// TIA Portal V19 export
FUNCTION "MFG TRANSFER CYCLE" : Void   // FC23, LAD
{ S7_Optimized_Access := 'TRUE' }
// stored: SetENOAutomatically false
   VAR_TEMP   // added for the SCL form of the ladder/FBD networks
      _w1 : Bool;
   END_VAR
BEGIN

REGION Network 1: TRANSFER SELECT
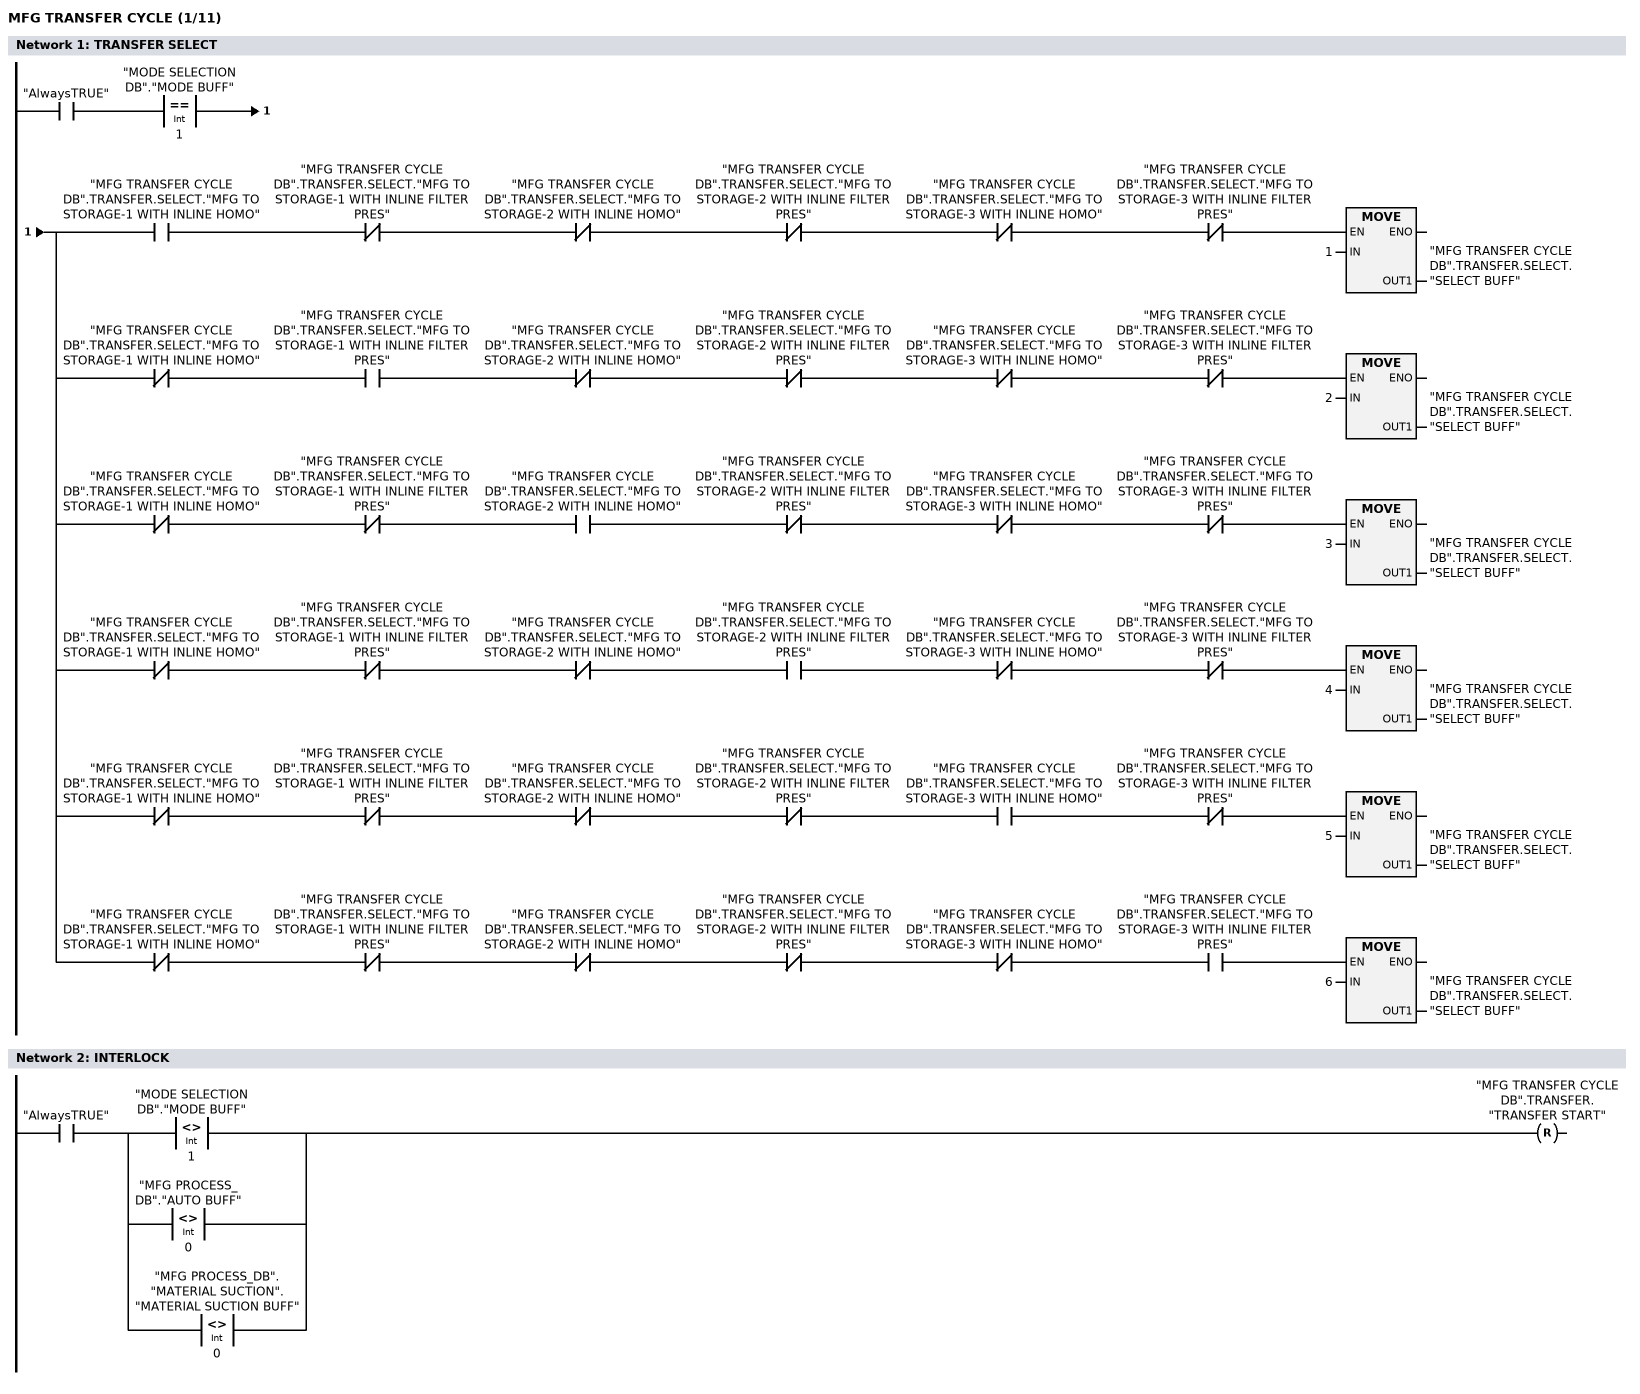
   RUNG wire#powerrail
      Contact( "AlwaysTRUE" )
      { S7_Templates := "SrcType := Int" } EQ_Contact(in1 := "MODE SELECTION DB"."MODE BUFF", in2 := 1)
      wire#w1
      Contact( "MFG TRANSFER CYCLE DB".TRANSFER.SELECT."MFG TO STORAGE-1 WITH INLINE HOMO" )
      I_Contact( "MFG TRANSFER CYCLE DB".TRANSFER.SELECT."MFG TO STORAGE-1 WITH INLINE FILTER PRES" )
      I_Contact( "MFG TRANSFER CYCLE DB".TRANSFER.SELECT."MFG TO STORAGE-2 WITH INLINE HOMO" )
      I_Contact( "MFG TRANSFER CYCLE DB".TRANSFER.SELECT."MFG TO STORAGE-2 WITH INLINE FILTER PRES" )
      I_Contact( "MFG TRANSFER CYCLE DB".TRANSFER.SELECT."MFG TO STORAGE-3 WITH INLINE HOMO" )
      I_Contact( "MFG TRANSFER CYCLE DB".TRANSFER.SELECT."MFG TO STORAGE-3 WITH INLINE FILTER PRES" )
      Move(in := 1, out1 => "MFG TRANSFER CYCLE DB".TRANSFER.SELECT."SELECT BUFF")
   END_RUNG
   RUNG wire#w1
      I_Contact( "MFG TRANSFER CYCLE DB".TRANSFER.SELECT."MFG TO STORAGE-1 WITH INLINE HOMO" )
      Contact( "MFG TRANSFER CYCLE DB".TRANSFER.SELECT."MFG TO STORAGE-1 WITH INLINE FILTER PRES" )
      I_Contact( "MFG TRANSFER CYCLE DB".TRANSFER.SELECT."MFG TO STORAGE-2 WITH INLINE HOMO" )
      I_Contact( "MFG TRANSFER CYCLE DB".TRANSFER.SELECT."MFG TO STORAGE-2 WITH INLINE FILTER PRES" )
      I_Contact( "MFG TRANSFER CYCLE DB".TRANSFER.SELECT."MFG TO STORAGE-3 WITH INLINE HOMO" )
      I_Contact( "MFG TRANSFER CYCLE DB".TRANSFER.SELECT."MFG TO STORAGE-3 WITH INLINE FILTER PRES" )
      Move(in := 2, out1 => "MFG TRANSFER CYCLE DB".TRANSFER.SELECT."SELECT BUFF")
   END_RUNG
   RUNG wire#w1
      I_Contact( "MFG TRANSFER CYCLE DB".TRANSFER.SELECT."MFG TO STORAGE-1 WITH INLINE HOMO" )
      I_Contact( "MFG TRANSFER CYCLE DB".TRANSFER.SELECT."MFG TO STORAGE-1 WITH INLINE FILTER PRES" )
      Contact( "MFG TRANSFER CYCLE DB".TRANSFER.SELECT."MFG TO STORAGE-2 WITH INLINE HOMO" )
      I_Contact( "MFG TRANSFER CYCLE DB".TRANSFER.SELECT."MFG TO STORAGE-2 WITH INLINE FILTER PRES" )
      I_Contact( "MFG TRANSFER CYCLE DB".TRANSFER.SELECT."MFG TO STORAGE-3 WITH INLINE HOMO" )
      I_Contact( "MFG TRANSFER CYCLE DB".TRANSFER.SELECT."MFG TO STORAGE-3 WITH INLINE FILTER PRES" )
      Move(in := 3, out1 => "MFG TRANSFER CYCLE DB".TRANSFER.SELECT."SELECT BUFF")
   END_RUNG
   RUNG wire#w1
      I_Contact( "MFG TRANSFER CYCLE DB".TRANSFER.SELECT."MFG TO STORAGE-1 WITH INLINE HOMO" )
      I_Contact( "MFG TRANSFER CYCLE DB".TRANSFER.SELECT."MFG TO STORAGE-1 WITH INLINE FILTER PRES" )
      I_Contact( "MFG TRANSFER CYCLE DB".TRANSFER.SELECT."MFG TO STORAGE-2 WITH INLINE HOMO" )
      Contact( "MFG TRANSFER CYCLE DB".TRANSFER.SELECT."MFG TO STORAGE-2 WITH INLINE FILTER PRES" )
      I_Contact( "MFG TRANSFER CYCLE DB".TRANSFER.SELECT."MFG TO STORAGE-3 WITH INLINE HOMO" )
      I_Contact( "MFG TRANSFER CYCLE DB".TRANSFER.SELECT."MFG TO STORAGE-3 WITH INLINE FILTER PRES" )
      Move(in := 4, out1 => "MFG TRANSFER CYCLE DB".TRANSFER.SELECT."SELECT BUFF")
   END_RUNG
   RUNG wire#w1
      I_Contact( "MFG TRANSFER CYCLE DB".TRANSFER.SELECT."MFG TO STORAGE-1 WITH INLINE HOMO" )
      I_Contact( "MFG TRANSFER CYCLE DB".TRANSFER.SELECT."MFG TO STORAGE-1 WITH INLINE FILTER PRES" )
      I_Contact( "MFG TRANSFER CYCLE DB".TRANSFER.SELECT."MFG TO STORAGE-2 WITH INLINE HOMO" )
      I_Contact( "MFG TRANSFER CYCLE DB".TRANSFER.SELECT."MFG TO STORAGE-2 WITH INLINE FILTER PRES" )
      Contact( "MFG TRANSFER CYCLE DB".TRANSFER.SELECT."MFG TO STORAGE-3 WITH INLINE HOMO" )
      I_Contact( "MFG TRANSFER CYCLE DB".TRANSFER.SELECT."MFG TO STORAGE-3 WITH INLINE FILTER PRES" )
      Move(in := 5, out1 => "MFG TRANSFER CYCLE DB".TRANSFER.SELECT."SELECT BUFF")
   END_RUNG
   RUNG wire#w1
      I_Contact( "MFG TRANSFER CYCLE DB".TRANSFER.SELECT."MFG TO STORAGE-1 WITH INLINE HOMO" )
      I_Contact( "MFG TRANSFER CYCLE DB".TRANSFER.SELECT."MFG TO STORAGE-1 WITH INLINE FILTER PRES" )
      I_Contact( "MFG TRANSFER CYCLE DB".TRANSFER.SELECT."MFG TO STORAGE-2 WITH INLINE HOMO" )
      I_Contact( "MFG TRANSFER CYCLE DB".TRANSFER.SELECT."MFG TO STORAGE-2 WITH INLINE FILTER PRES" )
      I_Contact( "MFG TRANSFER CYCLE DB".TRANSFER.SELECT."MFG TO STORAGE-3 WITH INLINE HOMO" )
      Contact( "MFG TRANSFER CYCLE DB".TRANSFER.SELECT."MFG TO STORAGE-3 WITH INLINE FILTER PRES" )
      Move(in := 6, out1 => "MFG TRANSFER CYCLE DB".TRANSFER.SELECT."SELECT BUFF")
   END_RUNG
   // the same network as SCL:
   #_w1 := "AlwaysTRUE" AND ("MODE SELECTION DB"."MODE BUFF" = 1);
   IF #_w1 AND "MFG TRANSFER CYCLE DB".TRANSFER.SELECT."MFG TO STORAGE-1 WITH INLINE HOMO" AND NOT "MFG TRANSFER CYCLE DB".TRANSFER.SELECT."MFG TO STORAGE-1 WITH INLINE FILTER PRES" AND NOT "MFG TRANSFER CYCLE DB".TRANSFER.SELECT."MFG TO STORAGE-2 WITH INLINE HOMO" AND NOT "MFG TRANSFER CYCLE DB".TRANSFER.SELECT."MFG TO STORAGE-2 WITH INLINE FILTER PRES" AND NOT "MFG TRANSFER CYCLE DB".TRANSFER.SELECT."MFG TO STORAGE-3 WITH INLINE HOMO" AND NOT "MFG TRANSFER CYCLE DB".TRANSFER.SELECT."MFG TO STORAGE-3 WITH INLINE FILTER PRES" THEN
       "MFG TRANSFER CYCLE DB".TRANSFER.SELECT."SELECT BUFF" := 1;
   END_IF;
   IF #_w1 AND NOT "MFG TRANSFER CYCLE DB".TRANSFER.SELECT."MFG TO STORAGE-1 WITH INLINE HOMO" AND "MFG TRANSFER CYCLE DB".TRANSFER.SELECT."MFG TO STORAGE-1 WITH INLINE FILTER PRES" AND NOT "MFG TRANSFER CYCLE DB".TRANSFER.SELECT."MFG TO STORAGE-2 WITH INLINE HOMO" AND NOT "MFG TRANSFER CYCLE DB".TRANSFER.SELECT."MFG TO STORAGE-2 WITH INLINE FILTER PRES" AND NOT "MFG TRANSFER CYCLE DB".TRANSFER.SELECT."MFG TO STORAGE-3 WITH INLINE HOMO" AND NOT "MFG TRANSFER CYCLE DB".TRANSFER.SELECT."MFG TO STORAGE-3 WITH INLINE FILTER PRES" THEN
       "MFG TRANSFER CYCLE DB".TRANSFER.SELECT."SELECT BUFF" := 2;
   END_IF;
   IF #_w1 AND NOT "MFG TRANSFER CYCLE DB".TRANSFER.SELECT."MFG TO STORAGE-1 WITH INLINE HOMO" AND NOT "MFG TRANSFER CYCLE DB".TRANSFER.SELECT."MFG TO STORAGE-1 WITH INLINE FILTER PRES" AND "MFG TRANSFER CYCLE DB".TRANSFER.SELECT."MFG TO STORAGE-2 WITH INLINE HOMO" AND NOT "MFG TRANSFER CYCLE DB".TRANSFER.SELECT."MFG TO STORAGE-2 WITH INLINE FILTER PRES" AND NOT "MFG TRANSFER CYCLE DB".TRANSFER.SELECT."MFG TO STORAGE-3 WITH INLINE HOMO" AND NOT "MFG TRANSFER CYCLE DB".TRANSFER.SELECT."MFG TO STORAGE-3 WITH INLINE FILTER PRES" THEN
       "MFG TRANSFER CYCLE DB".TRANSFER.SELECT."SELECT BUFF" := 3;
   END_IF;
   IF #_w1 AND NOT "MFG TRANSFER CYCLE DB".TRANSFER.SELECT."MFG TO STORAGE-1 WITH INLINE HOMO" AND NOT "MFG TRANSFER CYCLE DB".TRANSFER.SELECT."MFG TO STORAGE-1 WITH INLINE FILTER PRES" AND NOT "MFG TRANSFER CYCLE DB".TRANSFER.SELECT."MFG TO STORAGE-2 WITH INLINE HOMO" AND "MFG TRANSFER CYCLE DB".TRANSFER.SELECT."MFG TO STORAGE-2 WITH INLINE FILTER PRES" AND NOT "MFG TRANSFER CYCLE DB".TRANSFER.SELECT."MFG TO STORAGE-3 WITH INLINE HOMO" AND NOT "MFG TRANSFER CYCLE DB".TRANSFER.SELECT."MFG TO STORAGE-3 WITH INLINE FILTER PRES" THEN
       "MFG TRANSFER CYCLE DB".TRANSFER.SELECT."SELECT BUFF" := 4;
   END_IF;
   IF #_w1 AND NOT "MFG TRANSFER CYCLE DB".TRANSFER.SELECT."MFG TO STORAGE-1 WITH INLINE HOMO" AND NOT "MFG TRANSFER CYCLE DB".TRANSFER.SELECT."MFG TO STORAGE-1 WITH INLINE FILTER PRES" AND NOT "MFG TRANSFER CYCLE DB".TRANSFER.SELECT."MFG TO STORAGE-2 WITH INLINE HOMO" AND NOT "MFG TRANSFER CYCLE DB".TRANSFER.SELECT."MFG TO STORAGE-2 WITH INLINE FILTER PRES" AND "MFG TRANSFER CYCLE DB".TRANSFER.SELECT."MFG TO STORAGE-3 WITH INLINE HOMO" AND NOT "MFG TRANSFER CYCLE DB".TRANSFER.SELECT."MFG TO STORAGE-3 WITH INLINE FILTER PRES" THEN
       "MFG TRANSFER CYCLE DB".TRANSFER.SELECT."SELECT BUFF" := 5;
   END_IF;
   IF #_w1 AND NOT "MFG TRANSFER CYCLE DB".TRANSFER.SELECT."MFG TO STORAGE-1 WITH INLINE HOMO" AND NOT "MFG TRANSFER CYCLE DB".TRANSFER.SELECT."MFG TO STORAGE-1 WITH INLINE FILTER PRES" AND NOT "MFG TRANSFER CYCLE DB".TRANSFER.SELECT."MFG TO STORAGE-2 WITH INLINE HOMO" AND NOT "MFG TRANSFER CYCLE DB".TRANSFER.SELECT."MFG TO STORAGE-2 WITH INLINE FILTER PRES" AND NOT "MFG TRANSFER CYCLE DB".TRANSFER.SELECT."MFG TO STORAGE-3 WITH INLINE HOMO" AND "MFG TRANSFER CYCLE DB".TRANSFER.SELECT."MFG TO STORAGE-3 WITH INLINE FILTER PRES" THEN
       "MFG TRANSFER CYCLE DB".TRANSFER.SELECT."SELECT BUFF" := 6;
   END_IF;
END_REGION

REGION Network 2: INTERLOCK
   RUNG wire#powerrail
      Contact( "AlwaysTRUE" )
      wire#w1
      { S7_Templates := "SrcType := Int" } NE_Contact(in1 := "MODE SELECTION DB"."MODE BUFF", in2 := 1)
      wire#w2
      R_Coil( "MFG TRANSFER CYCLE DB".TRANSFER."TRANSFER START" )
   END_RUNG
   RUNG wire#w1
      { S7_Templates := "SrcType := Int" } NE_Contact(in1 := "MFG PROCESS_DB"."AUTO BUFF", in2 := 0)
   END_RUNG wire#w2
   RUNG wire#w1
      { S7_Templates := "SrcType := Int" } NE_Contact(in1 := "MFG PROCESS_DB"."MATERIAL SUCTION"."MATERIAL SUCTION BUFF", in2 := 0)
   END_RUNG wire#w2
   // the same network as SCL:
   IF "AlwaysTRUE" AND (("MODE SELECTION DB"."MODE BUFF" <> 1) OR ("MFG PROCESS_DB"."AUTO BUFF" <> 0) OR ("MFG PROCESS_DB"."MATERIAL SUCTION"."MATERIAL SUCTION BUFF" <> 0)) THEN
       "MFG TRANSFER CYCLE DB".TRANSFER."TRANSFER START" := FALSE;
   END_IF;
END_REGION

REGION Network 3: TRANSFER START ///////////////////////////// MFG TO STORAGE-1 WITH INLINE HOMO
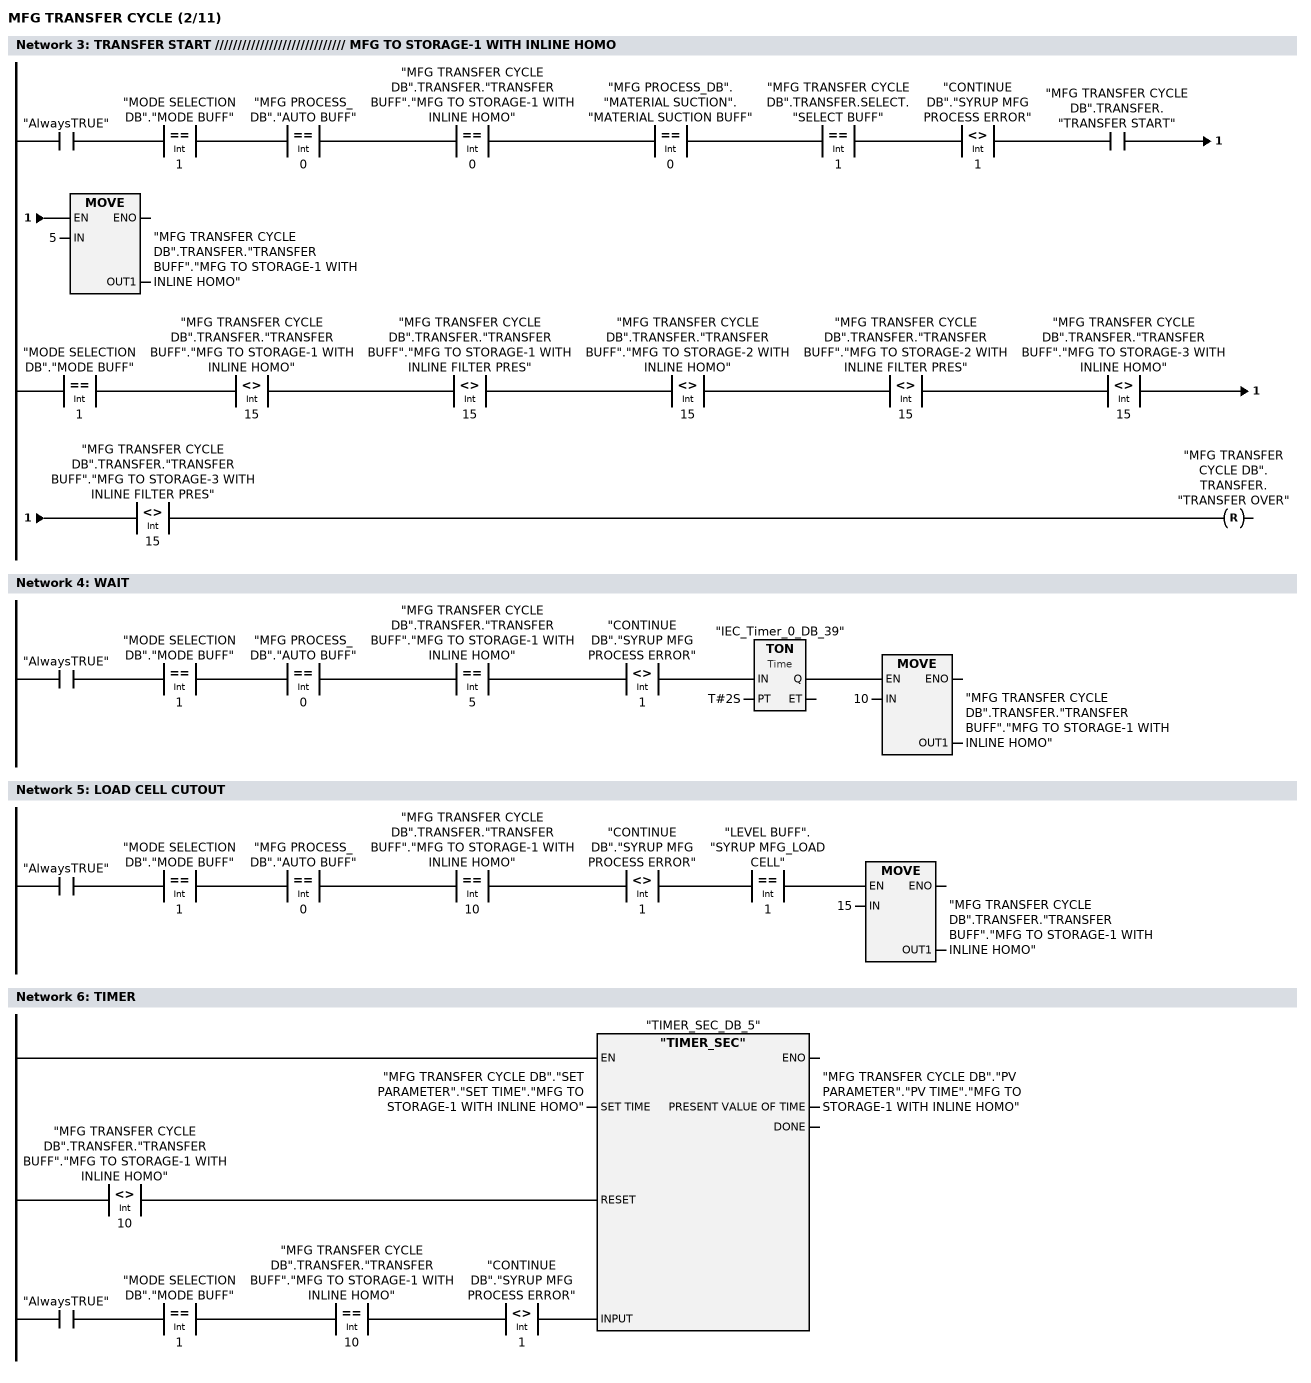
   RUNG wire#powerrail
      Contact( "AlwaysTRUE" )
      { S7_Templates := "SrcType := Int" } EQ_Contact(in1 := "MODE SELECTION DB"."MODE BUFF", in2 := 1)
      { S7_Templates := "SrcType := Int" } EQ_Contact(in1 := "MFG PROCESS_DB"."AUTO BUFF", in2 := 0)
      { S7_Templates := "SrcType := Int" } EQ_Contact(in1 := "MFG TRANSFER CYCLE DB".TRANSFER."TRANSFER BUFF"."MFG TO STORAGE-1 WITH INLINE HOMO", in2 := 0)
      { S7_Templates := "SrcType := Int" } EQ_Contact(in1 := "MFG PROCESS_DB"."MATERIAL SUCTION"."MATERIAL SUCTION BUFF", in2 := 0)
      { S7_Templates := "SrcType := Int" } EQ_Contact(in1 := "MFG TRANSFER CYCLE DB".TRANSFER.SELECT."SELECT BUFF", in2 := 1)
      { S7_Templates := "SrcType := Int" } NE_Contact(in1 := "CONTINUE DB"."SYRUP MFG PROCESS ERROR", in2 := 1)
      Contact( "MFG TRANSFER CYCLE DB".TRANSFER."TRANSFER START" )
      Move(in := 5, out1 => "MFG TRANSFER CYCLE DB".TRANSFER."TRANSFER BUFF"."MFG TO STORAGE-1 WITH INLINE HOMO")
   END_RUNG
   RUNG wire#powerrail
      { S7_Templates := "SrcType := Int" } EQ_Contact(in1 := "MODE SELECTION DB"."MODE BUFF", in2 := 1)
      { S7_Templates := "SrcType := Int" } NE_Contact(in1 := "MFG TRANSFER CYCLE DB".TRANSFER."TRANSFER BUFF"."MFG TO STORAGE-1 WITH INLINE HOMO", in2 := 15)
      { S7_Templates := "SrcType := Int" } NE_Contact(in1 := "MFG TRANSFER CYCLE DB".TRANSFER."TRANSFER BUFF"."MFG TO STORAGE-1 WITH INLINE FILTER PRES", in2 := 15)
      { S7_Templates := "SrcType := Int" } NE_Contact(in1 := "MFG TRANSFER CYCLE DB".TRANSFER."TRANSFER BUFF"."MFG TO STORAGE-2 WITH INLINE HOMO", in2 := 15)
      { S7_Templates := "SrcType := Int" } NE_Contact(in1 := "MFG TRANSFER CYCLE DB".TRANSFER."TRANSFER BUFF"."MFG TO STORAGE-2 WITH INLINE FILTER PRES", in2 := 15)
      { S7_Templates := "SrcType := Int" } NE_Contact(in1 := "MFG TRANSFER CYCLE DB".TRANSFER."TRANSFER BUFF"."MFG TO STORAGE-3 WITH INLINE HOMO", in2 := 15)
      { S7_Templates := "SrcType := Int" } NE_Contact(in1 := "MFG TRANSFER CYCLE DB".TRANSFER."TRANSFER BUFF"."MFG TO STORAGE-3 WITH INLINE FILTER PRES", in2 := 15)
      R_Coil( "MFG TRANSFER CYCLE DB".TRANSFER."TRANSFER OVER" )
   END_RUNG
   // the same network as SCL:
   IF "AlwaysTRUE" AND ("MODE SELECTION DB"."MODE BUFF" = 1) AND ("MFG PROCESS_DB"."AUTO BUFF" = 0) AND ("MFG TRANSFER CYCLE DB".TRANSFER."TRANSFER BUFF"."MFG TO STORAGE-1 WITH INLINE HOMO" = 0) AND ("MFG PROCESS_DB"."MATERIAL SUCTION"."MATERIAL SUCTION BUFF" = 0) AND ("MFG TRANSFER CYCLE DB".TRANSFER.SELECT."SELECT BUFF" = 1) AND ("CONTINUE DB"."SYRUP MFG PROCESS ERROR" <> 1) AND "MFG TRANSFER CYCLE DB".TRANSFER."TRANSFER START" THEN
       "MFG TRANSFER CYCLE DB".TRANSFER."TRANSFER BUFF"."MFG TO STORAGE-1 WITH INLINE HOMO" := 5;
   END_IF;
   IF ("MODE SELECTION DB"."MODE BUFF" = 1) AND ("MFG TRANSFER CYCLE DB".TRANSFER."TRANSFER BUFF"."MFG TO STORAGE-1 WITH INLINE HOMO" <> 15) AND ("MFG TRANSFER CYCLE DB".TRANSFER."TRANSFER BUFF"."MFG TO STORAGE-1 WITH INLINE FILTER PRES" <> 15) AND ("MFG TRANSFER CYCLE DB".TRANSFER."TRANSFER BUFF"."MFG TO STORAGE-2 WITH INLINE HOMO" <> 15) AND ("MFG TRANSFER CYCLE DB".TRANSFER."TRANSFER BUFF"."MFG TO STORAGE-2 WITH INLINE FILTER PRES" <> 15) AND ("MFG TRANSFER CYCLE DB".TRANSFER."TRANSFER BUFF"."MFG TO STORAGE-3 WITH INLINE HOMO" <> 15) AND ("MFG TRANSFER CYCLE DB".TRANSFER."TRANSFER BUFF"."MFG TO STORAGE-3 WITH INLINE FILTER PRES" <> 15) THEN
       "MFG TRANSFER CYCLE DB".TRANSFER."TRANSFER OVER" := FALSE;
   END_IF;
END_REGION

REGION Network 4: WAIT
   RUNG wire#powerrail
      Contact( "AlwaysTRUE" )
      { S7_Templates := "SrcType := Int" } EQ_Contact(in1 := "MODE SELECTION DB"."MODE BUFF", in2 := 1)
      { S7_Templates := "SrcType := Int" } EQ_Contact(in1 := "MFG PROCESS_DB"."AUTO BUFF", in2 := 0)
      { S7_Templates := "SrcType := Int" } EQ_Contact(in1 := "MFG TRANSFER CYCLE DB".TRANSFER."TRANSFER BUFF"."MFG TO STORAGE-1 WITH INLINE HOMO", in2 := 5)
      { S7_Templates := "SrcType := Int" } NE_Contact(in1 := "CONTINUE DB"."SYRUP MFG PROCESS ERROR", in2 := 1)
      { S7_Templates := "time_type := Time" } "IEC_Timer_0_DB_39".TON(pt := T#2S, et =>)
      Move(in := 10, out1 => "MFG TRANSFER CYCLE DB".TRANSFER."TRANSFER BUFF"."MFG TO STORAGE-1 WITH INLINE HOMO")
   END_RUNG
   // the same network as SCL:
   "IEC_Timer_0_DB_39".TON(IN := "AlwaysTRUE" AND ("MODE SELECTION DB"."MODE BUFF" = 1) AND ("MFG PROCESS_DB"."AUTO BUFF" = 0) AND ("MFG TRANSFER CYCLE DB".TRANSFER."TRANSFER BUFF"."MFG TO STORAGE-1 WITH INLINE HOMO" = 5) AND ("CONTINUE DB"."SYRUP MFG PROCESS ERROR" <> 1),
                           PT := T#2S);
   IF "IEC_Timer_0_DB_39".Q THEN
       "MFG TRANSFER CYCLE DB".TRANSFER."TRANSFER BUFF"."MFG TO STORAGE-1 WITH INLINE HOMO" := 10;
   END_IF;
END_REGION

REGION Network 5: LOAD CELL CUTOUT
   RUNG wire#powerrail
      Contact( "AlwaysTRUE" )
      { S7_Templates := "SrcType := Int" } EQ_Contact(in1 := "MODE SELECTION DB"."MODE BUFF", in2 := 1)
      { S7_Templates := "SrcType := Int" } EQ_Contact(in1 := "MFG PROCESS_DB"."AUTO BUFF", in2 := 0)
      { S7_Templates := "SrcType := Int" } EQ_Contact(in1 := "MFG TRANSFER CYCLE DB".TRANSFER."TRANSFER BUFF"."MFG TO STORAGE-1 WITH INLINE HOMO", in2 := 10)
      { S7_Templates := "SrcType := Int" } NE_Contact(in1 := "CONTINUE DB"."SYRUP MFG PROCESS ERROR", in2 := 1)
      { S7_Templates := "SrcType := Int" } EQ_Contact(in1 := "LEVEL BUFF"."SYRUP MFG_LOAD CELL", in2 := 1)
      Move(in := 15, out1 => "MFG TRANSFER CYCLE DB".TRANSFER."TRANSFER BUFF"."MFG TO STORAGE-1 WITH INLINE HOMO")
   END_RUNG
   // the same network as SCL:
   IF "AlwaysTRUE" AND ("MODE SELECTION DB"."MODE BUFF" = 1) AND ("MFG PROCESS_DB"."AUTO BUFF" = 0) AND ("MFG TRANSFER CYCLE DB".TRANSFER."TRANSFER BUFF"."MFG TO STORAGE-1 WITH INLINE HOMO" = 10) AND ("CONTINUE DB"."SYRUP MFG PROCESS ERROR" <> 1) AND ("LEVEL BUFF"."SYRUP MFG_LOAD CELL" = 1) THEN
       "MFG TRANSFER CYCLE DB".TRANSFER."TRANSFER BUFF"."MFG TO STORAGE-1 WITH INLINE HOMO" := 15;
   END_IF;
END_REGION

REGION Network 6: TIMER
   RUNG wire#powerrail
      "TIMER_SEC_DB_5"(RESET := wire#w1, INPUT := wire#w2, "SET TIME" := "MFG TRANSFER CYCLE DB"."SET PARAMETER"."SET TIME"."MFG TO STORAGE-1 WITH INLINE HOMO", "PRESENT VALUE OF TIME" => "MFG TRANSFER CYCLE DB"."PV PARAMETER"."PV TIME"."MFG TO STORAGE-1 WITH INLINE HOMO", DONE =>)
   END_RUNG
   RUNG wire#powerrail
      { S7_Templates := "SrcType := Int" } NE_Contact(in1 := "MFG TRANSFER CYCLE DB".TRANSFER."TRANSFER BUFF"."MFG TO STORAGE-1 WITH INLINE HOMO", in2 := 10)
   END_RUNG wire#w1
   RUNG wire#powerrail
      Contact( "AlwaysTRUE" )
      { S7_Templates := "SrcType := Int" } EQ_Contact(in1 := "MODE SELECTION DB"."MODE BUFF", in2 := 1)
      { S7_Templates := "SrcType := Int" } EQ_Contact(in1 := "MFG TRANSFER CYCLE DB".TRANSFER."TRANSFER BUFF"."MFG TO STORAGE-1 WITH INLINE HOMO", in2 := 10)
      { S7_Templates := "SrcType := Int" } NE_Contact(in1 := "CONTINUE DB"."SYRUP MFG PROCESS ERROR", in2 := 1)
   END_RUNG wire#w2
   // the same network as SCL:
   "TIMER_SEC_DB_5"("SET TIME" := "MFG TRANSFER CYCLE DB"."SET PARAMETER"."SET TIME"."MFG TO STORAGE-1 WITH INLINE HOMO",   // "TIMER_SEC"
                    RESET := "MFG TRANSFER CYCLE DB".TRANSFER."TRANSFER BUFF"."MFG TO STORAGE-1 WITH INLINE HOMO" <> 10,
                    INPUT := "AlwaysTRUE" AND ("MODE SELECTION DB"."MODE BUFF" = 1) AND ("MFG TRANSFER CYCLE DB".TRANSFER."TRANSFER BUFF"."MFG TO STORAGE-1 WITH INLINE HOMO" = 10) AND ("CONTINUE DB"."SYRUP MFG PROCESS ERROR" <> 1),
                    "PRESENT VALUE OF TIME" => "MFG TRANSFER CYCLE DB"."PV PARAMETER"."PV TIME"."MFG TO STORAGE-1 WITH INLINE HOMO");
END_REGION

REGION Network 7: TRANSFER OVER
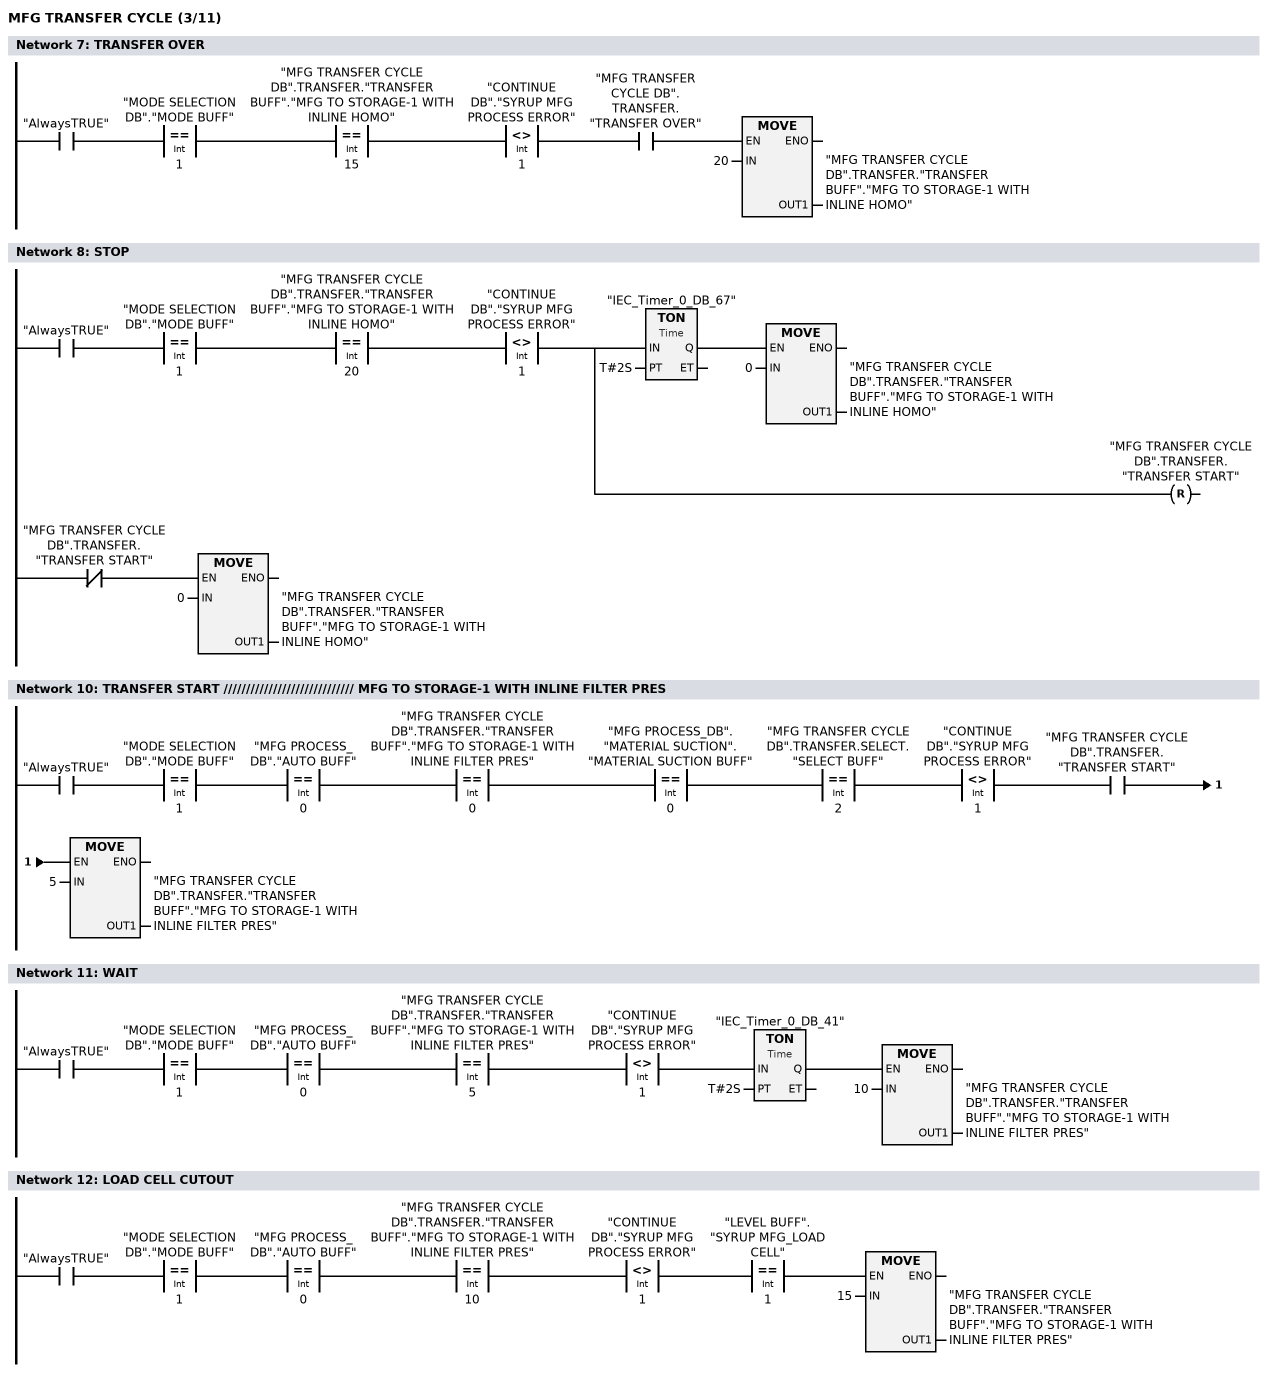
   RUNG wire#powerrail
      Contact( "AlwaysTRUE" )
      { S7_Templates := "SrcType := Int" } EQ_Contact(in1 := "MODE SELECTION DB"."MODE BUFF", in2 := 1)
      { S7_Templates := "SrcType := Int" } EQ_Contact(in1 := "MFG TRANSFER CYCLE DB".TRANSFER."TRANSFER BUFF"."MFG TO STORAGE-1 WITH INLINE HOMO", in2 := 15)
      { S7_Templates := "SrcType := Int" } NE_Contact(in1 := "CONTINUE DB"."SYRUP MFG PROCESS ERROR", in2 := 1)
      Contact( "MFG TRANSFER CYCLE DB".TRANSFER."TRANSFER OVER" )
      Move(in := 20, out1 => "MFG TRANSFER CYCLE DB".TRANSFER."TRANSFER BUFF"."MFG TO STORAGE-1 WITH INLINE HOMO")
   END_RUNG
   // the same network as SCL:
   IF "AlwaysTRUE" AND ("MODE SELECTION DB"."MODE BUFF" = 1) AND ("MFG TRANSFER CYCLE DB".TRANSFER."TRANSFER BUFF"."MFG TO STORAGE-1 WITH INLINE HOMO" = 15) AND ("CONTINUE DB"."SYRUP MFG PROCESS ERROR" <> 1) AND "MFG TRANSFER CYCLE DB".TRANSFER."TRANSFER OVER" THEN
       "MFG TRANSFER CYCLE DB".TRANSFER."TRANSFER BUFF"."MFG TO STORAGE-1 WITH INLINE HOMO" := 20;
   END_IF;
END_REGION

REGION Network 8: STOP
   RUNG wire#powerrail
      Contact( "AlwaysTRUE" )
      { S7_Templates := "SrcType := Int" } EQ_Contact(in1 := "MODE SELECTION DB"."MODE BUFF", in2 := 1)
      { S7_Templates := "SrcType := Int" } EQ_Contact(in1 := "MFG TRANSFER CYCLE DB".TRANSFER."TRANSFER BUFF"."MFG TO STORAGE-1 WITH INLINE HOMO", in2 := 20)
      { S7_Templates := "SrcType := Int" } NE_Contact(in1 := "CONTINUE DB"."SYRUP MFG PROCESS ERROR", in2 := 1)
      wire#w1
      { S7_Templates := "time_type := Time" } "IEC_Timer_0_DB_67".TON(pt := T#2S, et =>)
      Move(in := 0, out1 => "MFG TRANSFER CYCLE DB".TRANSFER."TRANSFER BUFF"."MFG TO STORAGE-1 WITH INLINE HOMO")
   END_RUNG
   RUNG wire#w1
      R_Coil( "MFG TRANSFER CYCLE DB".TRANSFER."TRANSFER START" )
   END_RUNG
   RUNG wire#powerrail
      I_Contact( "MFG TRANSFER CYCLE DB".TRANSFER."TRANSFER START" )
      Move(in := 0, out1 => "MFG TRANSFER CYCLE DB".TRANSFER."TRANSFER BUFF"."MFG TO STORAGE-1 WITH INLINE HOMO")
   END_RUNG
   // the same network as SCL:
   #_w1 := "AlwaysTRUE" AND ("MODE SELECTION DB"."MODE BUFF" = 1) AND ("MFG TRANSFER CYCLE DB".TRANSFER."TRANSFER BUFF"."MFG TO STORAGE-1 WITH INLINE HOMO" = 20) AND ("CONTINUE DB"."SYRUP MFG PROCESS ERROR" <> 1);
   "IEC_Timer_0_DB_67".TON(IN := #_w1, PT := T#2S);
   IF "IEC_Timer_0_DB_67".Q THEN
       "MFG TRANSFER CYCLE DB".TRANSFER."TRANSFER BUFF"."MFG TO STORAGE-1 WITH INLINE HOMO" := 0;
   END_IF;
   IF #_w1 THEN "MFG TRANSFER CYCLE DB".TRANSFER."TRANSFER START" := FALSE; END_IF;
   IF NOT "MFG TRANSFER CYCLE DB".TRANSFER."TRANSFER START" THEN
       "MFG TRANSFER CYCLE DB".TRANSFER."TRANSFER BUFF"."MFG TO STORAGE-1 WITH INLINE HOMO" := 0;
   END_IF;
END_REGION

REGION Network 10: TRANSFER START ///////////////////////////// MFG TO STORAGE-1 WITH INLINE FILTER PRES
   RUNG wire#powerrail
      Contact( "AlwaysTRUE" )
      { S7_Templates := "SrcType := Int" } EQ_Contact(in1 := "MODE SELECTION DB"."MODE BUFF", in2 := 1)
      { S7_Templates := "SrcType := Int" } EQ_Contact(in1 := "MFG PROCESS_DB"."AUTO BUFF", in2 := 0)
      { S7_Templates := "SrcType := Int" } EQ_Contact(in1 := "MFG TRANSFER CYCLE DB".TRANSFER."TRANSFER BUFF"."MFG TO STORAGE-1 WITH INLINE FILTER PRES", in2 := 0)
      { S7_Templates := "SrcType := Int" } EQ_Contact(in1 := "MFG PROCESS_DB"."MATERIAL SUCTION"."MATERIAL SUCTION BUFF", in2 := 0)
      { S7_Templates := "SrcType := Int" } EQ_Contact(in1 := "MFG TRANSFER CYCLE DB".TRANSFER.SELECT."SELECT BUFF", in2 := 2)
      { S7_Templates := "SrcType := Int" } NE_Contact(in1 := "CONTINUE DB"."SYRUP MFG PROCESS ERROR", in2 := 1)
      Contact( "MFG TRANSFER CYCLE DB".TRANSFER."TRANSFER START" )
      Move(in := 5, out1 => "MFG TRANSFER CYCLE DB".TRANSFER."TRANSFER BUFF"."MFG TO STORAGE-1 WITH INLINE FILTER PRES")
   END_RUNG
   // the same network as SCL:
   IF "AlwaysTRUE" AND ("MODE SELECTION DB"."MODE BUFF" = 1) AND ("MFG PROCESS_DB"."AUTO BUFF" = 0) AND ("MFG TRANSFER CYCLE DB".TRANSFER."TRANSFER BUFF"."MFG TO STORAGE-1 WITH INLINE FILTER PRES" = 0) AND ("MFG PROCESS_DB"."MATERIAL SUCTION"."MATERIAL SUCTION BUFF" = 0) AND ("MFG TRANSFER CYCLE DB".TRANSFER.SELECT."SELECT BUFF" = 2) AND ("CONTINUE DB"."SYRUP MFG PROCESS ERROR" <> 1) AND "MFG TRANSFER CYCLE DB".TRANSFER."TRANSFER START" THEN
       "MFG TRANSFER CYCLE DB".TRANSFER."TRANSFER BUFF"."MFG TO STORAGE-1 WITH INLINE FILTER PRES" := 5;
   END_IF;
END_REGION

REGION Network 11: WAIT
   RUNG wire#powerrail
      Contact( "AlwaysTRUE" )
      { S7_Templates := "SrcType := Int" } EQ_Contact(in1 := "MODE SELECTION DB"."MODE BUFF", in2 := 1)
      { S7_Templates := "SrcType := Int" } EQ_Contact(in1 := "MFG PROCESS_DB"."AUTO BUFF", in2 := 0)
      { S7_Templates := "SrcType := Int" } EQ_Contact(in1 := "MFG TRANSFER CYCLE DB".TRANSFER."TRANSFER BUFF"."MFG TO STORAGE-1 WITH INLINE FILTER PRES", in2 := 5)
      { S7_Templates := "SrcType := Int" } NE_Contact(in1 := "CONTINUE DB"."SYRUP MFG PROCESS ERROR", in2 := 1)
      { S7_Templates := "time_type := Time" } "IEC_Timer_0_DB_41".TON(pt := T#2S, et =>)
      Move(in := 10, out1 => "MFG TRANSFER CYCLE DB".TRANSFER."TRANSFER BUFF"."MFG TO STORAGE-1 WITH INLINE FILTER PRES")
   END_RUNG
   // the same network as SCL:
   "IEC_Timer_0_DB_41".TON(IN := "AlwaysTRUE" AND ("MODE SELECTION DB"."MODE BUFF" = 1) AND ("MFG PROCESS_DB"."AUTO BUFF" = 0) AND ("MFG TRANSFER CYCLE DB".TRANSFER."TRANSFER BUFF"."MFG TO STORAGE-1 WITH INLINE FILTER PRES" = 5) AND ("CONTINUE DB"."SYRUP MFG PROCESS ERROR" <> 1),
                           PT := T#2S);
   IF "IEC_Timer_0_DB_41".Q THEN
       "MFG TRANSFER CYCLE DB".TRANSFER."TRANSFER BUFF"."MFG TO STORAGE-1 WITH INLINE FILTER PRES" := 10;
   END_IF;
END_REGION

REGION Network 12: LOAD CELL CUTOUT
   RUNG wire#powerrail
      Contact( "AlwaysTRUE" )
      { S7_Templates := "SrcType := Int" } EQ_Contact(in1 := "MODE SELECTION DB"."MODE BUFF", in2 := 1)
      { S7_Templates := "SrcType := Int" } EQ_Contact(in1 := "MFG PROCESS_DB"."AUTO BUFF", in2 := 0)
      { S7_Templates := "SrcType := Int" } EQ_Contact(in1 := "MFG TRANSFER CYCLE DB".TRANSFER."TRANSFER BUFF"."MFG TO STORAGE-1 WITH INLINE FILTER PRES", in2 := 10)
      { S7_Templates := "SrcType := Int" } NE_Contact(in1 := "CONTINUE DB"."SYRUP MFG PROCESS ERROR", in2 := 1)
      { S7_Templates := "SrcType := Int" } EQ_Contact(in1 := "LEVEL BUFF"."SYRUP MFG_LOAD CELL", in2 := 1)
      Move(in := 15, out1 => "MFG TRANSFER CYCLE DB".TRANSFER."TRANSFER BUFF"."MFG TO STORAGE-1 WITH INLINE FILTER PRES")
   END_RUNG
   // the same network as SCL:
   IF "AlwaysTRUE" AND ("MODE SELECTION DB"."MODE BUFF" = 1) AND ("MFG PROCESS_DB"."AUTO BUFF" = 0) AND ("MFG TRANSFER CYCLE DB".TRANSFER."TRANSFER BUFF"."MFG TO STORAGE-1 WITH INLINE FILTER PRES" = 10) AND ("CONTINUE DB"."SYRUP MFG PROCESS ERROR" <> 1) AND ("LEVEL BUFF"."SYRUP MFG_LOAD CELL" = 1) THEN
       "MFG TRANSFER CYCLE DB".TRANSFER."TRANSFER BUFF"."MFG TO STORAGE-1 WITH INLINE FILTER PRES" := 15;
   END_IF;
END_REGION

REGION Network 13: TIMER
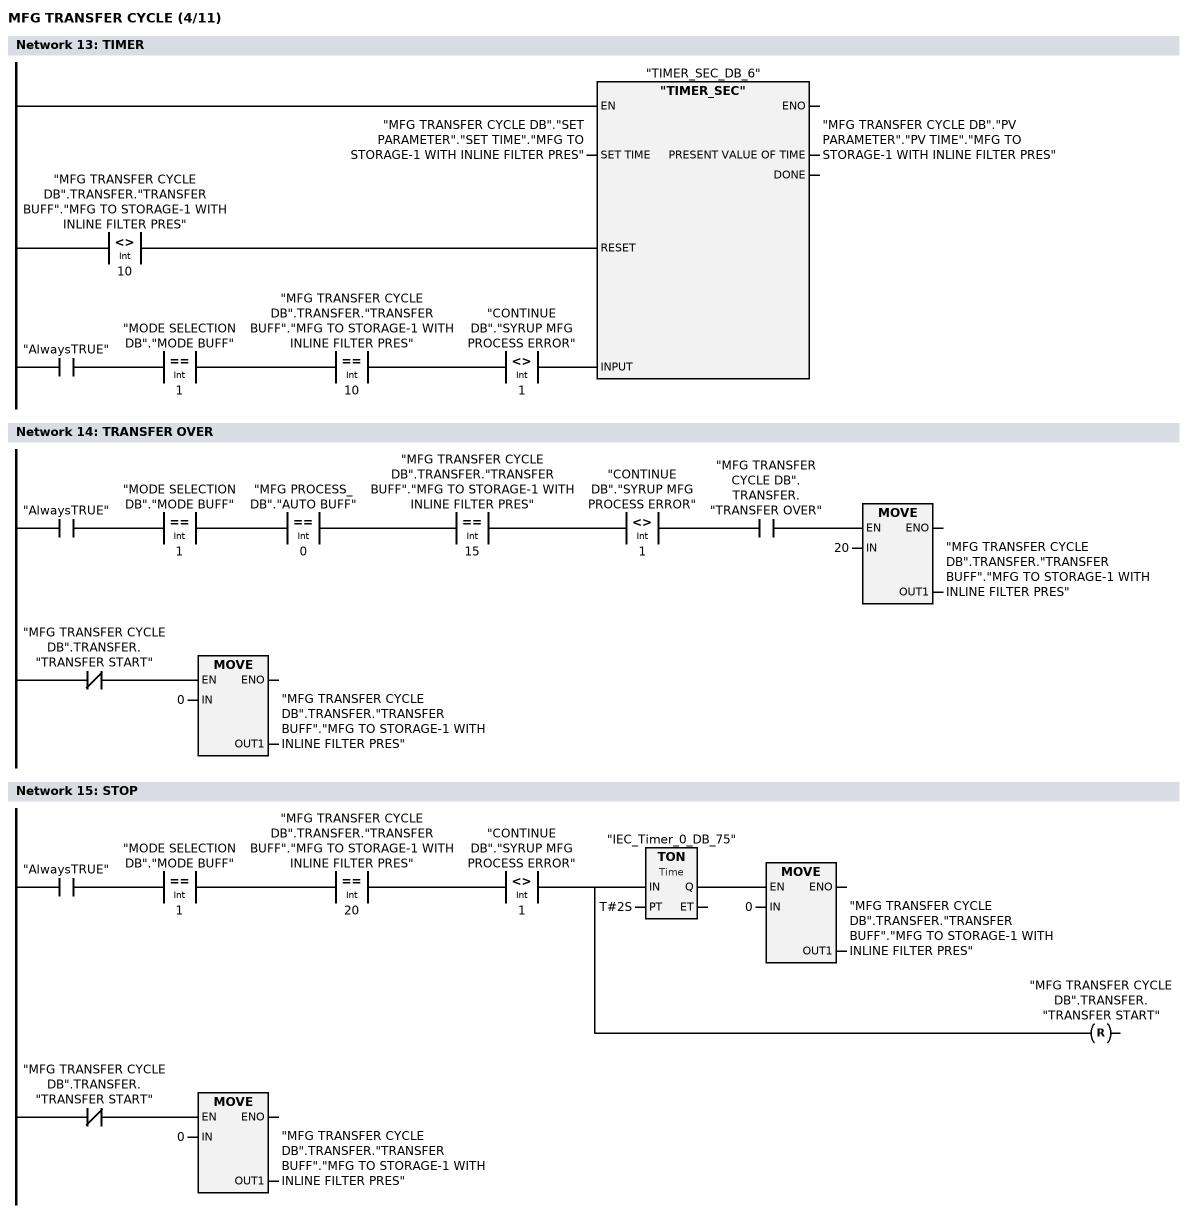
   RUNG wire#powerrail
      "TIMER_SEC_DB_6"(RESET := wire#w1, INPUT := wire#w2, "SET TIME" := "MFG TRANSFER CYCLE DB"."SET PARAMETER"."SET TIME"."MFG TO STORAGE-1 WITH INLINE FILTER PRES", "PRESENT VALUE OF TIME" => "MFG TRANSFER CYCLE DB"."PV PARAMETER"."PV TIME"."MFG TO STORAGE-1 WITH INLINE FILTER PRES", DONE =>)
   END_RUNG
   RUNG wire#powerrail
      { S7_Templates := "SrcType := Int" } NE_Contact(in1 := "MFG TRANSFER CYCLE DB".TRANSFER."TRANSFER BUFF"."MFG TO STORAGE-1 WITH INLINE FILTER PRES", in2 := 10)
   END_RUNG wire#w1
   RUNG wire#powerrail
      Contact( "AlwaysTRUE" )
      { S7_Templates := "SrcType := Int" } EQ_Contact(in1 := "MODE SELECTION DB"."MODE BUFF", in2 := 1)
      { S7_Templates := "SrcType := Int" } EQ_Contact(in1 := "MFG TRANSFER CYCLE DB".TRANSFER."TRANSFER BUFF"."MFG TO STORAGE-1 WITH INLINE FILTER PRES", in2 := 10)
      { S7_Templates := "SrcType := Int" } NE_Contact(in1 := "CONTINUE DB"."SYRUP MFG PROCESS ERROR", in2 := 1)
   END_RUNG wire#w2
   // the same network as SCL:
   "TIMER_SEC_DB_6"("SET TIME" := "MFG TRANSFER CYCLE DB"."SET PARAMETER"."SET TIME"."MFG TO STORAGE-1 WITH INLINE FILTER PRES",   // "TIMER_SEC"
                    RESET := "MFG TRANSFER CYCLE DB".TRANSFER."TRANSFER BUFF"."MFG TO STORAGE-1 WITH INLINE FILTER PRES" <> 10,
                    INPUT := "AlwaysTRUE" AND ("MODE SELECTION DB"."MODE BUFF" = 1) AND ("MFG TRANSFER CYCLE DB".TRANSFER."TRANSFER BUFF"."MFG TO STORAGE-1 WITH INLINE FILTER PRES" = 10) AND ("CONTINUE DB"."SYRUP MFG PROCESS ERROR" <> 1),
                    "PRESENT VALUE OF TIME" => "MFG TRANSFER CYCLE DB"."PV PARAMETER"."PV TIME"."MFG TO STORAGE-1 WITH INLINE FILTER PRES");
END_REGION

REGION Network 14: TRANSFER OVER
   RUNG wire#powerrail
      Contact( "AlwaysTRUE" )
      { S7_Templates := "SrcType := Int" } EQ_Contact(in1 := "MODE SELECTION DB"."MODE BUFF", in2 := 1)
      { S7_Templates := "SrcType := Int" } EQ_Contact(in1 := "MFG PROCESS_DB"."AUTO BUFF", in2 := 0)
      { S7_Templates := "SrcType := Int" } EQ_Contact(in1 := "MFG TRANSFER CYCLE DB".TRANSFER."TRANSFER BUFF"."MFG TO STORAGE-1 WITH INLINE FILTER PRES", in2 := 15)
      { S7_Templates := "SrcType := Int" } NE_Contact(in1 := "CONTINUE DB"."SYRUP MFG PROCESS ERROR", in2 := 1)
      Contact( "MFG TRANSFER CYCLE DB".TRANSFER."TRANSFER OVER" )
      Move(in := 20, out1 => "MFG TRANSFER CYCLE DB".TRANSFER."TRANSFER BUFF"."MFG TO STORAGE-1 WITH INLINE FILTER PRES")
   END_RUNG
   RUNG wire#powerrail
      I_Contact( "MFG TRANSFER CYCLE DB".TRANSFER."TRANSFER START" )
      Move(in := 0, out1 => "MFG TRANSFER CYCLE DB".TRANSFER."TRANSFER BUFF"."MFG TO STORAGE-1 WITH INLINE FILTER PRES")
   END_RUNG
   // the same network as SCL:
   IF "AlwaysTRUE" AND ("MODE SELECTION DB"."MODE BUFF" = 1) AND ("MFG PROCESS_DB"."AUTO BUFF" = 0) AND ("MFG TRANSFER CYCLE DB".TRANSFER."TRANSFER BUFF"."MFG TO STORAGE-1 WITH INLINE FILTER PRES" = 15) AND ("CONTINUE DB"."SYRUP MFG PROCESS ERROR" <> 1) AND "MFG TRANSFER CYCLE DB".TRANSFER."TRANSFER OVER" THEN
       "MFG TRANSFER CYCLE DB".TRANSFER."TRANSFER BUFF"."MFG TO STORAGE-1 WITH INLINE FILTER PRES" := 20;
   END_IF;
   IF NOT "MFG TRANSFER CYCLE DB".TRANSFER."TRANSFER START" THEN
       "MFG TRANSFER CYCLE DB".TRANSFER."TRANSFER BUFF"."MFG TO STORAGE-1 WITH INLINE FILTER PRES" := 0;
   END_IF;
END_REGION

REGION Network 15: STOP
   RUNG wire#powerrail
      Contact( "AlwaysTRUE" )
      { S7_Templates := "SrcType := Int" } EQ_Contact(in1 := "MODE SELECTION DB"."MODE BUFF", in2 := 1)
      { S7_Templates := "SrcType := Int" } EQ_Contact(in1 := "MFG TRANSFER CYCLE DB".TRANSFER."TRANSFER BUFF"."MFG TO STORAGE-1 WITH INLINE FILTER PRES", in2 := 20)
      { S7_Templates := "SrcType := Int" } NE_Contact(in1 := "CONTINUE DB"."SYRUP MFG PROCESS ERROR", in2 := 1)
      wire#w1
      { S7_Templates := "time_type := Time" } "IEC_Timer_0_DB_75".TON(pt := T#2S, et =>)
      Move(in := 0, out1 => "MFG TRANSFER CYCLE DB".TRANSFER."TRANSFER BUFF"."MFG TO STORAGE-1 WITH INLINE FILTER PRES")
   END_RUNG
   RUNG wire#w1
      R_Coil( "MFG TRANSFER CYCLE DB".TRANSFER."TRANSFER START" )
   END_RUNG
   RUNG wire#powerrail
      I_Contact( "MFG TRANSFER CYCLE DB".TRANSFER."TRANSFER START" )
      Move(in := 0, out1 => "MFG TRANSFER CYCLE DB".TRANSFER."TRANSFER BUFF"."MFG TO STORAGE-1 WITH INLINE FILTER PRES")
   END_RUNG
   // the same network as SCL:
   #_w1 := "AlwaysTRUE" AND ("MODE SELECTION DB"."MODE BUFF" = 1) AND ("MFG TRANSFER CYCLE DB".TRANSFER."TRANSFER BUFF"."MFG TO STORAGE-1 WITH INLINE FILTER PRES" = 20) AND ("CONTINUE DB"."SYRUP MFG PROCESS ERROR" <> 1);
   "IEC_Timer_0_DB_75".TON(IN := #_w1, PT := T#2S);
   IF "IEC_Timer_0_DB_75".Q THEN
       "MFG TRANSFER CYCLE DB".TRANSFER."TRANSFER BUFF"."MFG TO STORAGE-1 WITH INLINE FILTER PRES" := 0;
   END_IF;
   IF #_w1 THEN "MFG TRANSFER CYCLE DB".TRANSFER."TRANSFER START" := FALSE; END_IF;
   IF NOT "MFG TRANSFER CYCLE DB".TRANSFER."TRANSFER START" THEN
       "MFG TRANSFER CYCLE DB".TRANSFER."TRANSFER BUFF"."MFG TO STORAGE-1 WITH INLINE FILTER PRES" := 0;
   END_IF;
END_REGION

REGION Network 17: TRANSFER START ///////////////////////////// MFG TO STORAGE-2 WITH INLINE HOMO
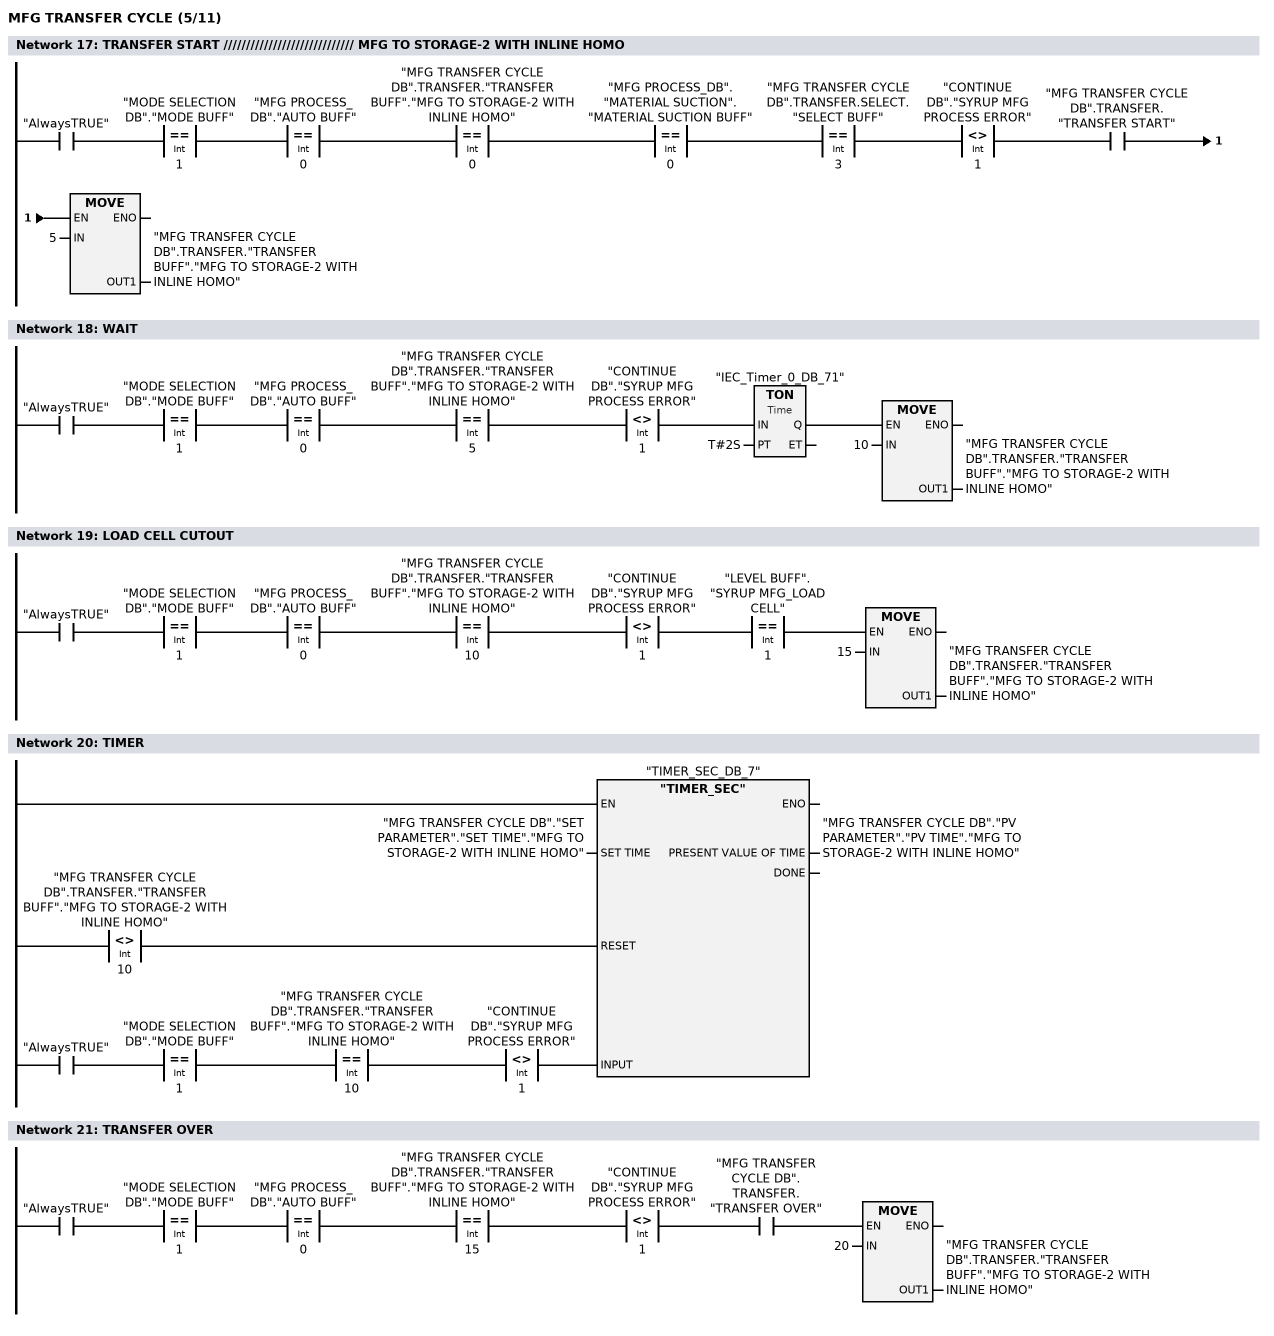
   RUNG wire#powerrail
      Contact( "AlwaysTRUE" )
      { S7_Templates := "SrcType := Int" } EQ_Contact(in1 := "MODE SELECTION DB"."MODE BUFF", in2 := 1)
      { S7_Templates := "SrcType := Int" } EQ_Contact(in1 := "MFG PROCESS_DB"."AUTO BUFF", in2 := 0)
      { S7_Templates := "SrcType := Int" } EQ_Contact(in1 := "MFG TRANSFER CYCLE DB".TRANSFER."TRANSFER BUFF"."MFG TO STORAGE-2 WITH INLINE HOMO", in2 := 0)
      { S7_Templates := "SrcType := Int" } EQ_Contact(in1 := "MFG PROCESS_DB"."MATERIAL SUCTION"."MATERIAL SUCTION BUFF", in2 := 0)
      { S7_Templates := "SrcType := Int" } EQ_Contact(in1 := "MFG TRANSFER CYCLE DB".TRANSFER.SELECT."SELECT BUFF", in2 := 3)
      { S7_Templates := "SrcType := Int" } NE_Contact(in1 := "CONTINUE DB"."SYRUP MFG PROCESS ERROR", in2 := 1)
      Contact( "MFG TRANSFER CYCLE DB".TRANSFER."TRANSFER START" )
      Move(in := 5, out1 => "MFG TRANSFER CYCLE DB".TRANSFER."TRANSFER BUFF"."MFG TO STORAGE-2 WITH INLINE HOMO")
   END_RUNG
   // the same network as SCL:
   IF "AlwaysTRUE" AND ("MODE SELECTION DB"."MODE BUFF" = 1) AND ("MFG PROCESS_DB"."AUTO BUFF" = 0) AND ("MFG TRANSFER CYCLE DB".TRANSFER."TRANSFER BUFF"."MFG TO STORAGE-2 WITH INLINE HOMO" = 0) AND ("MFG PROCESS_DB"."MATERIAL SUCTION"."MATERIAL SUCTION BUFF" = 0) AND ("MFG TRANSFER CYCLE DB".TRANSFER.SELECT."SELECT BUFF" = 3) AND ("CONTINUE DB"."SYRUP MFG PROCESS ERROR" <> 1) AND "MFG TRANSFER CYCLE DB".TRANSFER."TRANSFER START" THEN
       "MFG TRANSFER CYCLE DB".TRANSFER."TRANSFER BUFF"."MFG TO STORAGE-2 WITH INLINE HOMO" := 5;
   END_IF;
END_REGION

REGION Network 18: WAIT
   RUNG wire#powerrail
      Contact( "AlwaysTRUE" )
      { S7_Templates := "SrcType := Int" } EQ_Contact(in1 := "MODE SELECTION DB"."MODE BUFF", in2 := 1)
      { S7_Templates := "SrcType := Int" } EQ_Contact(in1 := "MFG PROCESS_DB"."AUTO BUFF", in2 := 0)
      { S7_Templates := "SrcType := Int" } EQ_Contact(in1 := "MFG TRANSFER CYCLE DB".TRANSFER."TRANSFER BUFF"."MFG TO STORAGE-2 WITH INLINE HOMO", in2 := 5)
      { S7_Templates := "SrcType := Int" } NE_Contact(in1 := "CONTINUE DB"."SYRUP MFG PROCESS ERROR", in2 := 1)
      { S7_Templates := "time_type := Time" } "IEC_Timer_0_DB_71".TON(pt := T#2S, et =>)
      Move(in := 10, out1 => "MFG TRANSFER CYCLE DB".TRANSFER."TRANSFER BUFF"."MFG TO STORAGE-2 WITH INLINE HOMO")
   END_RUNG
   // the same network as SCL:
   "IEC_Timer_0_DB_71".TON(IN := "AlwaysTRUE" AND ("MODE SELECTION DB"."MODE BUFF" = 1) AND ("MFG PROCESS_DB"."AUTO BUFF" = 0) AND ("MFG TRANSFER CYCLE DB".TRANSFER."TRANSFER BUFF"."MFG TO STORAGE-2 WITH INLINE HOMO" = 5) AND ("CONTINUE DB"."SYRUP MFG PROCESS ERROR" <> 1),
                           PT := T#2S);
   IF "IEC_Timer_0_DB_71".Q THEN
       "MFG TRANSFER CYCLE DB".TRANSFER."TRANSFER BUFF"."MFG TO STORAGE-2 WITH INLINE HOMO" := 10;
   END_IF;
END_REGION

REGION Network 19: LOAD CELL CUTOUT
   RUNG wire#powerrail
      Contact( "AlwaysTRUE" )
      { S7_Templates := "SrcType := Int" } EQ_Contact(in1 := "MODE SELECTION DB"."MODE BUFF", in2 := 1)
      { S7_Templates := "SrcType := Int" } EQ_Contact(in1 := "MFG PROCESS_DB"."AUTO BUFF", in2 := 0)
      { S7_Templates := "SrcType := Int" } EQ_Contact(in1 := "MFG TRANSFER CYCLE DB".TRANSFER."TRANSFER BUFF"."MFG TO STORAGE-2 WITH INLINE HOMO", in2 := 10)
      { S7_Templates := "SrcType := Int" } NE_Contact(in1 := "CONTINUE DB"."SYRUP MFG PROCESS ERROR", in2 := 1)
      { S7_Templates := "SrcType := Int" } EQ_Contact(in1 := "LEVEL BUFF"."SYRUP MFG_LOAD CELL", in2 := 1)
      Move(in := 15, out1 => "MFG TRANSFER CYCLE DB".TRANSFER."TRANSFER BUFF"."MFG TO STORAGE-2 WITH INLINE HOMO")
   END_RUNG
   // the same network as SCL:
   IF "AlwaysTRUE" AND ("MODE SELECTION DB"."MODE BUFF" = 1) AND ("MFG PROCESS_DB"."AUTO BUFF" = 0) AND ("MFG TRANSFER CYCLE DB".TRANSFER."TRANSFER BUFF"."MFG TO STORAGE-2 WITH INLINE HOMO" = 10) AND ("CONTINUE DB"."SYRUP MFG PROCESS ERROR" <> 1) AND ("LEVEL BUFF"."SYRUP MFG_LOAD CELL" = 1) THEN
       "MFG TRANSFER CYCLE DB".TRANSFER."TRANSFER BUFF"."MFG TO STORAGE-2 WITH INLINE HOMO" := 15;
   END_IF;
END_REGION

REGION Network 20: TIMER
   RUNG wire#powerrail
      "TIMER_SEC_DB_7"(RESET := wire#w1, INPUT := wire#w2, "SET TIME" := "MFG TRANSFER CYCLE DB"."SET PARAMETER"."SET TIME"."MFG TO STORAGE-2 WITH INLINE HOMO", "PRESENT VALUE OF TIME" => "MFG TRANSFER CYCLE DB"."PV PARAMETER"."PV TIME"."MFG TO STORAGE-2 WITH INLINE HOMO", DONE =>)
   END_RUNG
   RUNG wire#powerrail
      { S7_Templates := "SrcType := Int" } NE_Contact(in1 := "MFG TRANSFER CYCLE DB".TRANSFER."TRANSFER BUFF"."MFG TO STORAGE-2 WITH INLINE HOMO", in2 := 10)
   END_RUNG wire#w1
   RUNG wire#powerrail
      Contact( "AlwaysTRUE" )
      { S7_Templates := "SrcType := Int" } EQ_Contact(in1 := "MODE SELECTION DB"."MODE BUFF", in2 := 1)
      { S7_Templates := "SrcType := Int" } EQ_Contact(in1 := "MFG TRANSFER CYCLE DB".TRANSFER."TRANSFER BUFF"."MFG TO STORAGE-2 WITH INLINE HOMO", in2 := 10)
      { S7_Templates := "SrcType := Int" } NE_Contact(in1 := "CONTINUE DB"."SYRUP MFG PROCESS ERROR", in2 := 1)
   END_RUNG wire#w2
   // the same network as SCL:
   "TIMER_SEC_DB_7"("SET TIME" := "MFG TRANSFER CYCLE DB"."SET PARAMETER"."SET TIME"."MFG TO STORAGE-2 WITH INLINE HOMO",   // "TIMER_SEC"
                    RESET := "MFG TRANSFER CYCLE DB".TRANSFER."TRANSFER BUFF"."MFG TO STORAGE-2 WITH INLINE HOMO" <> 10,
                    INPUT := "AlwaysTRUE" AND ("MODE SELECTION DB"."MODE BUFF" = 1) AND ("MFG TRANSFER CYCLE DB".TRANSFER."TRANSFER BUFF"."MFG TO STORAGE-2 WITH INLINE HOMO" = 10) AND ("CONTINUE DB"."SYRUP MFG PROCESS ERROR" <> 1),
                    "PRESENT VALUE OF TIME" => "MFG TRANSFER CYCLE DB"."PV PARAMETER"."PV TIME"."MFG TO STORAGE-2 WITH INLINE HOMO");
END_REGION

REGION Network 21: TRANSFER OVER
   RUNG wire#powerrail
      Contact( "AlwaysTRUE" )
      { S7_Templates := "SrcType := Int" } EQ_Contact(in1 := "MODE SELECTION DB"."MODE BUFF", in2 := 1)
      { S7_Templates := "SrcType := Int" } EQ_Contact(in1 := "MFG PROCESS_DB"."AUTO BUFF", in2 := 0)
      { S7_Templates := "SrcType := Int" } EQ_Contact(in1 := "MFG TRANSFER CYCLE DB".TRANSFER."TRANSFER BUFF"."MFG TO STORAGE-2 WITH INLINE HOMO", in2 := 15)
      { S7_Templates := "SrcType := Int" } NE_Contact(in1 := "CONTINUE DB"."SYRUP MFG PROCESS ERROR", in2 := 1)
      Contact( "MFG TRANSFER CYCLE DB".TRANSFER."TRANSFER OVER" )
      Move(in := 20, out1 => "MFG TRANSFER CYCLE DB".TRANSFER."TRANSFER BUFF"."MFG TO STORAGE-2 WITH INLINE HOMO")
   END_RUNG
   // the same network as SCL:
   IF "AlwaysTRUE" AND ("MODE SELECTION DB"."MODE BUFF" = 1) AND ("MFG PROCESS_DB"."AUTO BUFF" = 0) AND ("MFG TRANSFER CYCLE DB".TRANSFER."TRANSFER BUFF"."MFG TO STORAGE-2 WITH INLINE HOMO" = 15) AND ("CONTINUE DB"."SYRUP MFG PROCESS ERROR" <> 1) AND "MFG TRANSFER CYCLE DB".TRANSFER."TRANSFER OVER" THEN
       "MFG TRANSFER CYCLE DB".TRANSFER."TRANSFER BUFF"."MFG TO STORAGE-2 WITH INLINE HOMO" := 20;
   END_IF;
END_REGION

REGION Network 22: STOP
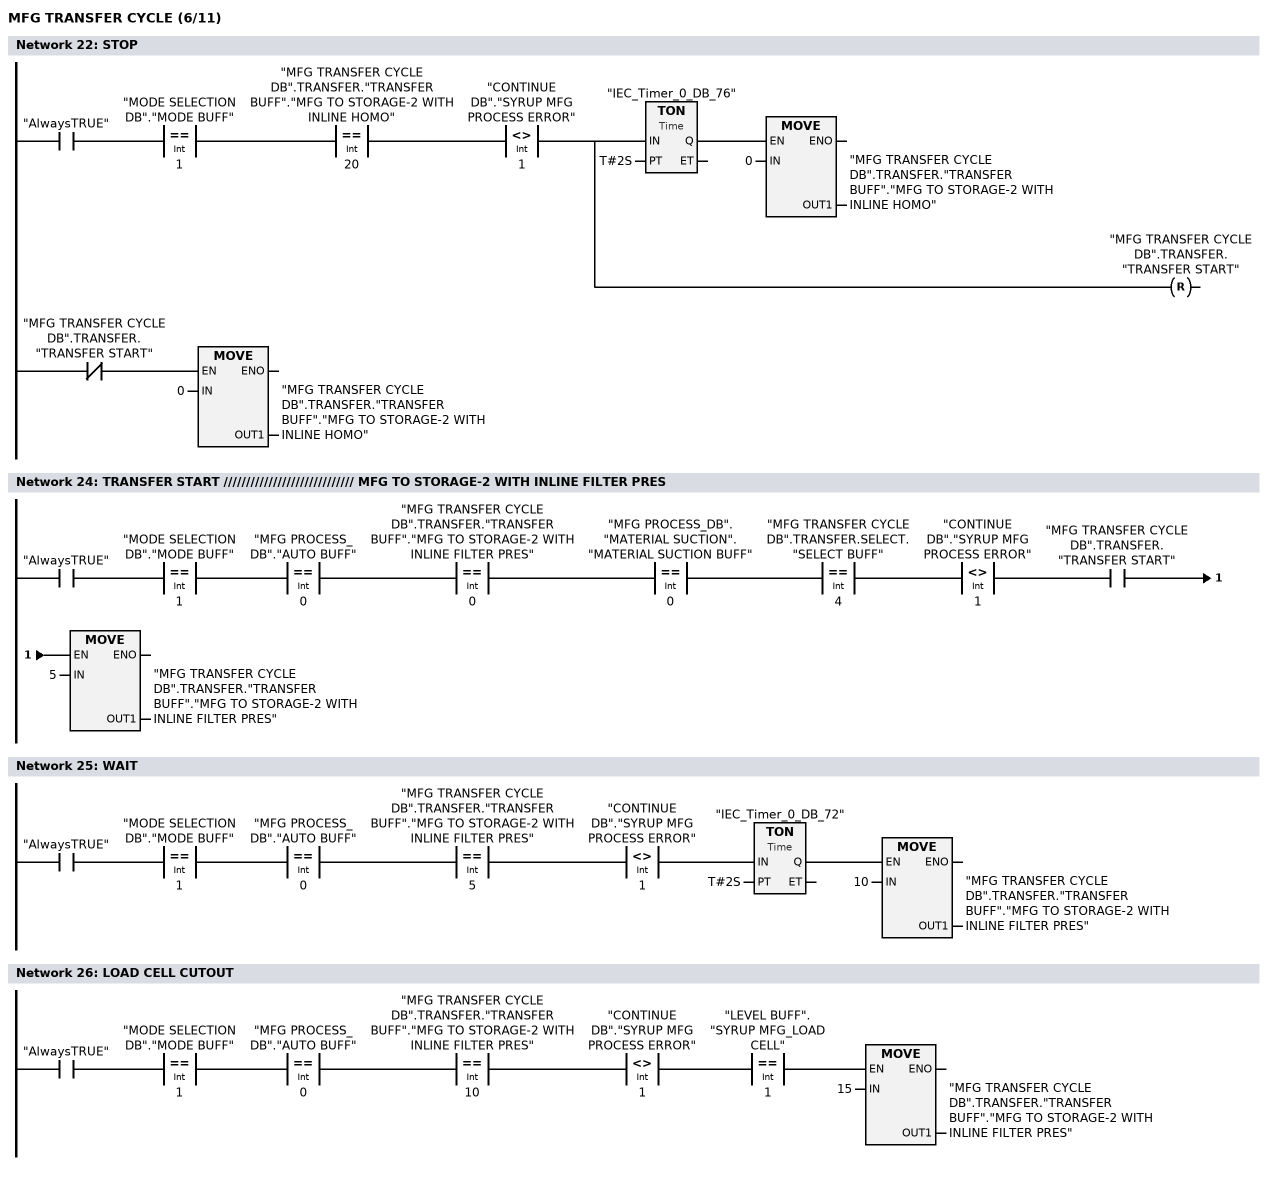
   RUNG wire#powerrail
      Contact( "AlwaysTRUE" )
      { S7_Templates := "SrcType := Int" } EQ_Contact(in1 := "MODE SELECTION DB"."MODE BUFF", in2 := 1)
      { S7_Templates := "SrcType := Int" } EQ_Contact(in1 := "MFG TRANSFER CYCLE DB".TRANSFER."TRANSFER BUFF"."MFG TO STORAGE-2 WITH INLINE HOMO", in2 := 20)
      { S7_Templates := "SrcType := Int" } NE_Contact(in1 := "CONTINUE DB"."SYRUP MFG PROCESS ERROR", in2 := 1)
      wire#w1
      { S7_Templates := "time_type := Time" } "IEC_Timer_0_DB_76".TON(pt := T#2S, et =>)
      Move(in := 0, out1 => "MFG TRANSFER CYCLE DB".TRANSFER."TRANSFER BUFF"."MFG TO STORAGE-2 WITH INLINE HOMO")
   END_RUNG
   RUNG wire#w1
      R_Coil( "MFG TRANSFER CYCLE DB".TRANSFER."TRANSFER START" )
   END_RUNG
   RUNG wire#powerrail
      I_Contact( "MFG TRANSFER CYCLE DB".TRANSFER."TRANSFER START" )
      Move(in := 0, out1 => "MFG TRANSFER CYCLE DB".TRANSFER."TRANSFER BUFF"."MFG TO STORAGE-2 WITH INLINE HOMO")
   END_RUNG
   // the same network as SCL:
   #_w1 := "AlwaysTRUE" AND ("MODE SELECTION DB"."MODE BUFF" = 1) AND ("MFG TRANSFER CYCLE DB".TRANSFER."TRANSFER BUFF"."MFG TO STORAGE-2 WITH INLINE HOMO" = 20) AND ("CONTINUE DB"."SYRUP MFG PROCESS ERROR" <> 1);
   "IEC_Timer_0_DB_76".TON(IN := #_w1, PT := T#2S);
   IF "IEC_Timer_0_DB_76".Q THEN
       "MFG TRANSFER CYCLE DB".TRANSFER."TRANSFER BUFF"."MFG TO STORAGE-2 WITH INLINE HOMO" := 0;
   END_IF;
   IF #_w1 THEN "MFG TRANSFER CYCLE DB".TRANSFER."TRANSFER START" := FALSE; END_IF;
   IF NOT "MFG TRANSFER CYCLE DB".TRANSFER."TRANSFER START" THEN
       "MFG TRANSFER CYCLE DB".TRANSFER."TRANSFER BUFF"."MFG TO STORAGE-2 WITH INLINE HOMO" := 0;
   END_IF;
END_REGION

REGION Network 24: TRANSFER START ///////////////////////////// MFG TO STORAGE-2 WITH INLINE FILTER PRES
   RUNG wire#powerrail
      Contact( "AlwaysTRUE" )
      { S7_Templates := "SrcType := Int" } EQ_Contact(in1 := "MODE SELECTION DB"."MODE BUFF", in2 := 1)
      { S7_Templates := "SrcType := Int" } EQ_Contact(in1 := "MFG PROCESS_DB"."AUTO BUFF", in2 := 0)
      { S7_Templates := "SrcType := Int" } EQ_Contact(in1 := "MFG TRANSFER CYCLE DB".TRANSFER."TRANSFER BUFF"."MFG TO STORAGE-2 WITH INLINE FILTER PRES", in2 := 0)
      { S7_Templates := "SrcType := Int" } EQ_Contact(in1 := "MFG PROCESS_DB"."MATERIAL SUCTION"."MATERIAL SUCTION BUFF", in2 := 0)
      { S7_Templates := "SrcType := Int" } EQ_Contact(in1 := "MFG TRANSFER CYCLE DB".TRANSFER.SELECT."SELECT BUFF", in2 := 4)
      { S7_Templates := "SrcType := Int" } NE_Contact(in1 := "CONTINUE DB"."SYRUP MFG PROCESS ERROR", in2 := 1)
      Contact( "MFG TRANSFER CYCLE DB".TRANSFER."TRANSFER START" )
      Move(in := 5, out1 => "MFG TRANSFER CYCLE DB".TRANSFER."TRANSFER BUFF"."MFG TO STORAGE-2 WITH INLINE FILTER PRES")
   END_RUNG
   // the same network as SCL:
   IF "AlwaysTRUE" AND ("MODE SELECTION DB"."MODE BUFF" = 1) AND ("MFG PROCESS_DB"."AUTO BUFF" = 0) AND ("MFG TRANSFER CYCLE DB".TRANSFER."TRANSFER BUFF"."MFG TO STORAGE-2 WITH INLINE FILTER PRES" = 0) AND ("MFG PROCESS_DB"."MATERIAL SUCTION"."MATERIAL SUCTION BUFF" = 0) AND ("MFG TRANSFER CYCLE DB".TRANSFER.SELECT."SELECT BUFF" = 4) AND ("CONTINUE DB"."SYRUP MFG PROCESS ERROR" <> 1) AND "MFG TRANSFER CYCLE DB".TRANSFER."TRANSFER START" THEN
       "MFG TRANSFER CYCLE DB".TRANSFER."TRANSFER BUFF"."MFG TO STORAGE-2 WITH INLINE FILTER PRES" := 5;
   END_IF;
END_REGION

REGION Network 25: WAIT
   RUNG wire#powerrail
      Contact( "AlwaysTRUE" )
      { S7_Templates := "SrcType := Int" } EQ_Contact(in1 := "MODE SELECTION DB"."MODE BUFF", in2 := 1)
      { S7_Templates := "SrcType := Int" } EQ_Contact(in1 := "MFG PROCESS_DB"."AUTO BUFF", in2 := 0)
      { S7_Templates := "SrcType := Int" } EQ_Contact(in1 := "MFG TRANSFER CYCLE DB".TRANSFER."TRANSFER BUFF"."MFG TO STORAGE-2 WITH INLINE FILTER PRES", in2 := 5)
      { S7_Templates := "SrcType := Int" } NE_Contact(in1 := "CONTINUE DB"."SYRUP MFG PROCESS ERROR", in2 := 1)
      { S7_Templates := "time_type := Time" } "IEC_Timer_0_DB_72".TON(pt := T#2S, et =>)
      Move(in := 10, out1 => "MFG TRANSFER CYCLE DB".TRANSFER."TRANSFER BUFF"."MFG TO STORAGE-2 WITH INLINE FILTER PRES")
   END_RUNG
   // the same network as SCL:
   "IEC_Timer_0_DB_72".TON(IN := "AlwaysTRUE" AND ("MODE SELECTION DB"."MODE BUFF" = 1) AND ("MFG PROCESS_DB"."AUTO BUFF" = 0) AND ("MFG TRANSFER CYCLE DB".TRANSFER."TRANSFER BUFF"."MFG TO STORAGE-2 WITH INLINE FILTER PRES" = 5) AND ("CONTINUE DB"."SYRUP MFG PROCESS ERROR" <> 1),
                           PT := T#2S);
   IF "IEC_Timer_0_DB_72".Q THEN
       "MFG TRANSFER CYCLE DB".TRANSFER."TRANSFER BUFF"."MFG TO STORAGE-2 WITH INLINE FILTER PRES" := 10;
   END_IF;
END_REGION

REGION Network 26: LOAD CELL CUTOUT
   RUNG wire#powerrail
      Contact( "AlwaysTRUE" )
      { S7_Templates := "SrcType := Int" } EQ_Contact(in1 := "MODE SELECTION DB"."MODE BUFF", in2 := 1)
      { S7_Templates := "SrcType := Int" } EQ_Contact(in1 := "MFG PROCESS_DB"."AUTO BUFF", in2 := 0)
      { S7_Templates := "SrcType := Int" } EQ_Contact(in1 := "MFG TRANSFER CYCLE DB".TRANSFER."TRANSFER BUFF"."MFG TO STORAGE-2 WITH INLINE FILTER PRES", in2 := 10)
      { S7_Templates := "SrcType := Int" } NE_Contact(in1 := "CONTINUE DB"."SYRUP MFG PROCESS ERROR", in2 := 1)
      { S7_Templates := "SrcType := Int" } EQ_Contact(in1 := "LEVEL BUFF"."SYRUP MFG_LOAD CELL", in2 := 1)
      Move(in := 15, out1 => "MFG TRANSFER CYCLE DB".TRANSFER."TRANSFER BUFF"."MFG TO STORAGE-2 WITH INLINE FILTER PRES")
   END_RUNG
   // the same network as SCL:
   IF "AlwaysTRUE" AND ("MODE SELECTION DB"."MODE BUFF" = 1) AND ("MFG PROCESS_DB"."AUTO BUFF" = 0) AND ("MFG TRANSFER CYCLE DB".TRANSFER."TRANSFER BUFF"."MFG TO STORAGE-2 WITH INLINE FILTER PRES" = 10) AND ("CONTINUE DB"."SYRUP MFG PROCESS ERROR" <> 1) AND ("LEVEL BUFF"."SYRUP MFG_LOAD CELL" = 1) THEN
       "MFG TRANSFER CYCLE DB".TRANSFER."TRANSFER BUFF"."MFG TO STORAGE-2 WITH INLINE FILTER PRES" := 15;
   END_IF;
END_REGION

REGION Network 27: TIMER
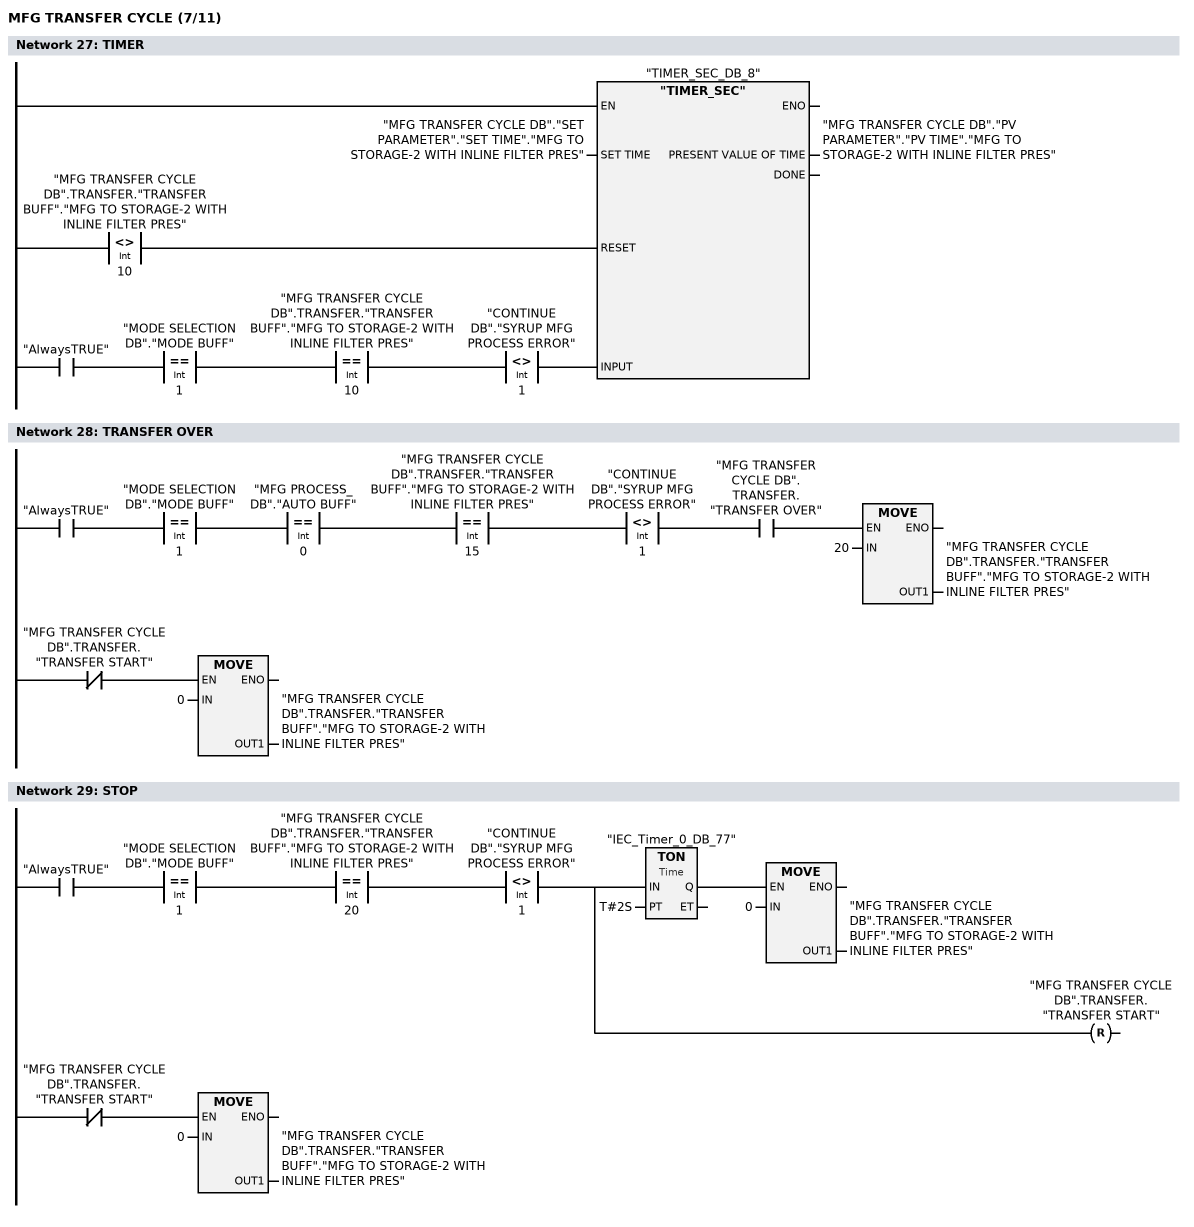
   RUNG wire#powerrail
      "TIMER_SEC_DB_8"(RESET := wire#w1, INPUT := wire#w2, "SET TIME" := "MFG TRANSFER CYCLE DB"."SET PARAMETER"."SET TIME"."MFG TO STORAGE-2 WITH INLINE FILTER PRES", "PRESENT VALUE OF TIME" => "MFG TRANSFER CYCLE DB"."PV PARAMETER"."PV TIME"."MFG TO STORAGE-2 WITH INLINE FILTER PRES", DONE =>)
   END_RUNG
   RUNG wire#powerrail
      { S7_Templates := "SrcType := Int" } NE_Contact(in1 := "MFG TRANSFER CYCLE DB".TRANSFER."TRANSFER BUFF"."MFG TO STORAGE-2 WITH INLINE FILTER PRES", in2 := 10)
   END_RUNG wire#w1
   RUNG wire#powerrail
      Contact( "AlwaysTRUE" )
      { S7_Templates := "SrcType := Int" } EQ_Contact(in1 := "MODE SELECTION DB"."MODE BUFF", in2 := 1)
      { S7_Templates := "SrcType := Int" } EQ_Contact(in1 := "MFG TRANSFER CYCLE DB".TRANSFER."TRANSFER BUFF"."MFG TO STORAGE-2 WITH INLINE FILTER PRES", in2 := 10)
      { S7_Templates := "SrcType := Int" } NE_Contact(in1 := "CONTINUE DB"."SYRUP MFG PROCESS ERROR", in2 := 1)
   END_RUNG wire#w2
   // the same network as SCL:
   "TIMER_SEC_DB_8"("SET TIME" := "MFG TRANSFER CYCLE DB"."SET PARAMETER"."SET TIME"."MFG TO STORAGE-2 WITH INLINE FILTER PRES",   // "TIMER_SEC"
                    RESET := "MFG TRANSFER CYCLE DB".TRANSFER."TRANSFER BUFF"."MFG TO STORAGE-2 WITH INLINE FILTER PRES" <> 10,
                    INPUT := "AlwaysTRUE" AND ("MODE SELECTION DB"."MODE BUFF" = 1) AND ("MFG TRANSFER CYCLE DB".TRANSFER."TRANSFER BUFF"."MFG TO STORAGE-2 WITH INLINE FILTER PRES" = 10) AND ("CONTINUE DB"."SYRUP MFG PROCESS ERROR" <> 1),
                    "PRESENT VALUE OF TIME" => "MFG TRANSFER CYCLE DB"."PV PARAMETER"."PV TIME"."MFG TO STORAGE-2 WITH INLINE FILTER PRES");
END_REGION

REGION Network 28: TRANSFER OVER
   RUNG wire#powerrail
      Contact( "AlwaysTRUE" )
      { S7_Templates := "SrcType := Int" } EQ_Contact(in1 := "MODE SELECTION DB"."MODE BUFF", in2 := 1)
      { S7_Templates := "SrcType := Int" } EQ_Contact(in1 := "MFG PROCESS_DB"."AUTO BUFF", in2 := 0)
      { S7_Templates := "SrcType := Int" } EQ_Contact(in1 := "MFG TRANSFER CYCLE DB".TRANSFER."TRANSFER BUFF"."MFG TO STORAGE-2 WITH INLINE FILTER PRES", in2 := 15)
      { S7_Templates := "SrcType := Int" } NE_Contact(in1 := "CONTINUE DB"."SYRUP MFG PROCESS ERROR", in2 := 1)
      Contact( "MFG TRANSFER CYCLE DB".TRANSFER."TRANSFER OVER" )
      Move(in := 20, out1 => "MFG TRANSFER CYCLE DB".TRANSFER."TRANSFER BUFF"."MFG TO STORAGE-2 WITH INLINE FILTER PRES")
   END_RUNG
   RUNG wire#powerrail
      I_Contact( "MFG TRANSFER CYCLE DB".TRANSFER."TRANSFER START" )
      Move(in := 0, out1 => "MFG TRANSFER CYCLE DB".TRANSFER."TRANSFER BUFF"."MFG TO STORAGE-2 WITH INLINE FILTER PRES")
   END_RUNG
   // the same network as SCL:
   IF "AlwaysTRUE" AND ("MODE SELECTION DB"."MODE BUFF" = 1) AND ("MFG PROCESS_DB"."AUTO BUFF" = 0) AND ("MFG TRANSFER CYCLE DB".TRANSFER."TRANSFER BUFF"."MFG TO STORAGE-2 WITH INLINE FILTER PRES" = 15) AND ("CONTINUE DB"."SYRUP MFG PROCESS ERROR" <> 1) AND "MFG TRANSFER CYCLE DB".TRANSFER."TRANSFER OVER" THEN
       "MFG TRANSFER CYCLE DB".TRANSFER."TRANSFER BUFF"."MFG TO STORAGE-2 WITH INLINE FILTER PRES" := 20;
   END_IF;
   IF NOT "MFG TRANSFER CYCLE DB".TRANSFER."TRANSFER START" THEN
       "MFG TRANSFER CYCLE DB".TRANSFER."TRANSFER BUFF"."MFG TO STORAGE-2 WITH INLINE FILTER PRES" := 0;
   END_IF;
END_REGION

REGION Network 29: STOP
   RUNG wire#powerrail
      Contact( "AlwaysTRUE" )
      { S7_Templates := "SrcType := Int" } EQ_Contact(in1 := "MODE SELECTION DB"."MODE BUFF", in2 := 1)
      { S7_Templates := "SrcType := Int" } EQ_Contact(in1 := "MFG TRANSFER CYCLE DB".TRANSFER."TRANSFER BUFF"."MFG TO STORAGE-2 WITH INLINE FILTER PRES", in2 := 20)
      { S7_Templates := "SrcType := Int" } NE_Contact(in1 := "CONTINUE DB"."SYRUP MFG PROCESS ERROR", in2 := 1)
      wire#w1
      { S7_Templates := "time_type := Time" } "IEC_Timer_0_DB_77".TON(pt := T#2S, et =>)
      Move(in := 0, out1 => "MFG TRANSFER CYCLE DB".TRANSFER."TRANSFER BUFF"."MFG TO STORAGE-2 WITH INLINE FILTER PRES")
   END_RUNG
   RUNG wire#w1
      R_Coil( "MFG TRANSFER CYCLE DB".TRANSFER."TRANSFER START" )
   END_RUNG
   RUNG wire#powerrail
      I_Contact( "MFG TRANSFER CYCLE DB".TRANSFER."TRANSFER START" )
      Move(in := 0, out1 => "MFG TRANSFER CYCLE DB".TRANSFER."TRANSFER BUFF"."MFG TO STORAGE-2 WITH INLINE FILTER PRES")
   END_RUNG
   // the same network as SCL:
   #_w1 := "AlwaysTRUE" AND ("MODE SELECTION DB"."MODE BUFF" = 1) AND ("MFG TRANSFER CYCLE DB".TRANSFER."TRANSFER BUFF"."MFG TO STORAGE-2 WITH INLINE FILTER PRES" = 20) AND ("CONTINUE DB"."SYRUP MFG PROCESS ERROR" <> 1);
   "IEC_Timer_0_DB_77".TON(IN := #_w1, PT := T#2S);
   IF "IEC_Timer_0_DB_77".Q THEN
       "MFG TRANSFER CYCLE DB".TRANSFER."TRANSFER BUFF"."MFG TO STORAGE-2 WITH INLINE FILTER PRES" := 0;
   END_IF;
   IF #_w1 THEN "MFG TRANSFER CYCLE DB".TRANSFER."TRANSFER START" := FALSE; END_IF;
   IF NOT "MFG TRANSFER CYCLE DB".TRANSFER."TRANSFER START" THEN
       "MFG TRANSFER CYCLE DB".TRANSFER."TRANSFER BUFF"."MFG TO STORAGE-2 WITH INLINE FILTER PRES" := 0;
   END_IF;
END_REGION

REGION Network 31: TRANSFER START ///////////////////////////// MFG TO STORAGE-3 WITH INLINE HOMO
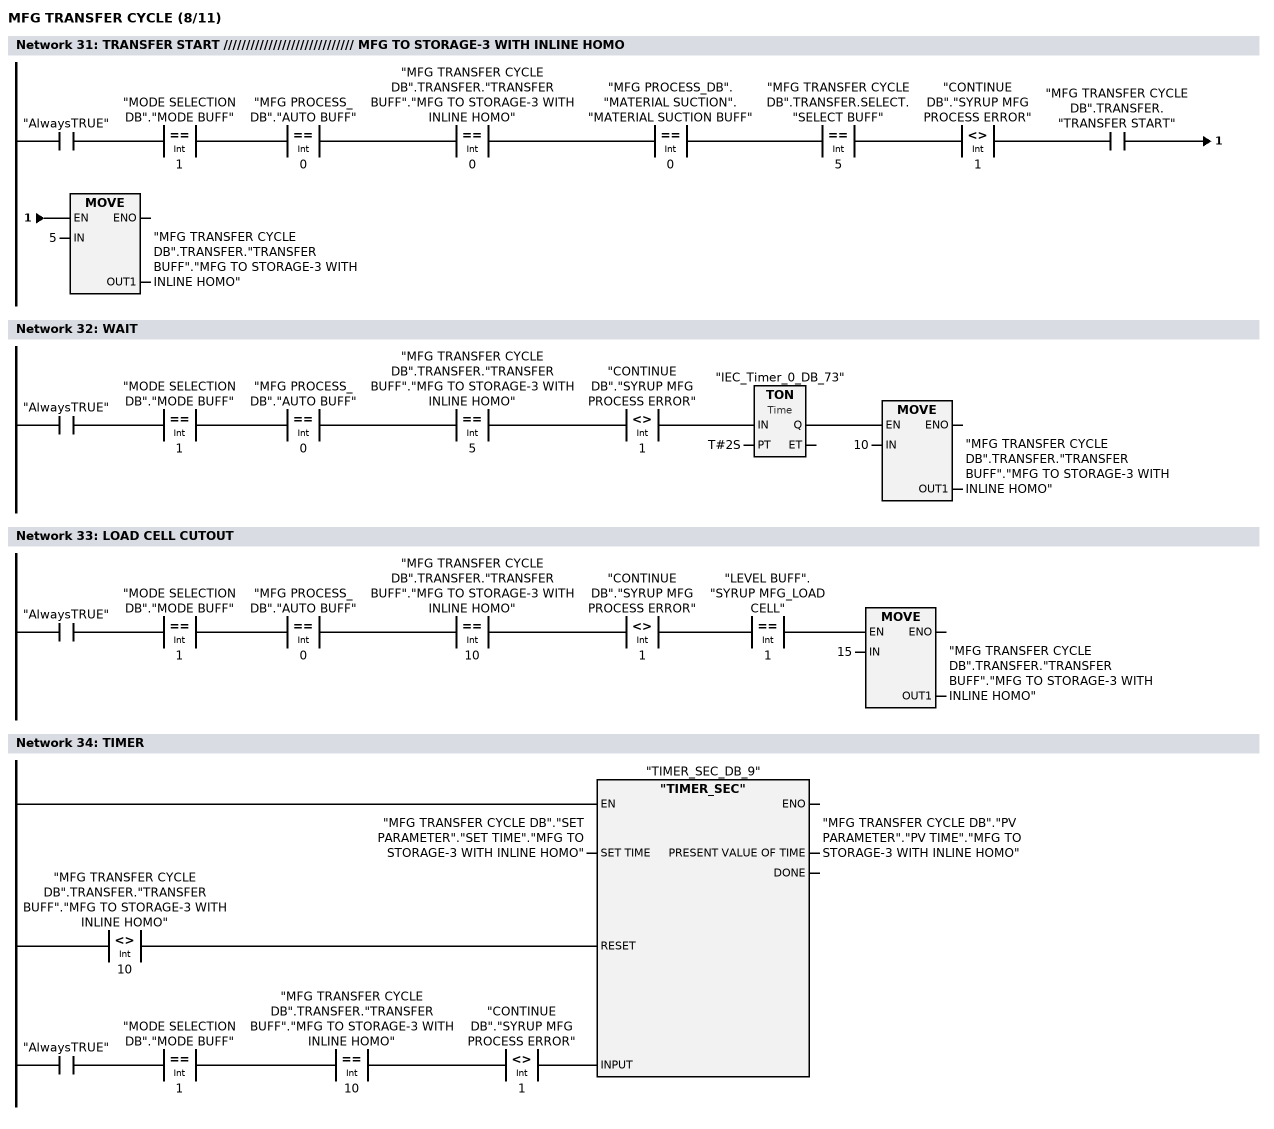
   RUNG wire#powerrail
      Contact( "AlwaysTRUE" )
      { S7_Templates := "SrcType := Int" } EQ_Contact(in1 := "MODE SELECTION DB"."MODE BUFF", in2 := 1)
      { S7_Templates := "SrcType := Int" } EQ_Contact(in1 := "MFG PROCESS_DB"."AUTO BUFF", in2 := 0)
      { S7_Templates := "SrcType := Int" } EQ_Contact(in1 := "MFG TRANSFER CYCLE DB".TRANSFER."TRANSFER BUFF"."MFG TO STORAGE-3 WITH INLINE HOMO", in2 := 0)
      { S7_Templates := "SrcType := Int" } EQ_Contact(in1 := "MFG PROCESS_DB"."MATERIAL SUCTION"."MATERIAL SUCTION BUFF", in2 := 0)
      { S7_Templates := "SrcType := Int" } EQ_Contact(in1 := "MFG TRANSFER CYCLE DB".TRANSFER.SELECT."SELECT BUFF", in2 := 5)
      { S7_Templates := "SrcType := Int" } NE_Contact(in1 := "CONTINUE DB"."SYRUP MFG PROCESS ERROR", in2 := 1)
      Contact( "MFG TRANSFER CYCLE DB".TRANSFER."TRANSFER START" )
      Move(in := 5, out1 => "MFG TRANSFER CYCLE DB".TRANSFER."TRANSFER BUFF"."MFG TO STORAGE-3 WITH INLINE HOMO")
   END_RUNG
   // the same network as SCL:
   IF "AlwaysTRUE" AND ("MODE SELECTION DB"."MODE BUFF" = 1) AND ("MFG PROCESS_DB"."AUTO BUFF" = 0) AND ("MFG TRANSFER CYCLE DB".TRANSFER."TRANSFER BUFF"."MFG TO STORAGE-3 WITH INLINE HOMO" = 0) AND ("MFG PROCESS_DB"."MATERIAL SUCTION"."MATERIAL SUCTION BUFF" = 0) AND ("MFG TRANSFER CYCLE DB".TRANSFER.SELECT."SELECT BUFF" = 5) AND ("CONTINUE DB"."SYRUP MFG PROCESS ERROR" <> 1) AND "MFG TRANSFER CYCLE DB".TRANSFER."TRANSFER START" THEN
       "MFG TRANSFER CYCLE DB".TRANSFER."TRANSFER BUFF"."MFG TO STORAGE-3 WITH INLINE HOMO" := 5;
   END_IF;
END_REGION

REGION Network 32: WAIT
   RUNG wire#powerrail
      Contact( "AlwaysTRUE" )
      { S7_Templates := "SrcType := Int" } EQ_Contact(in1 := "MODE SELECTION DB"."MODE BUFF", in2 := 1)
      { S7_Templates := "SrcType := Int" } EQ_Contact(in1 := "MFG PROCESS_DB"."AUTO BUFF", in2 := 0)
      { S7_Templates := "SrcType := Int" } EQ_Contact(in1 := "MFG TRANSFER CYCLE DB".TRANSFER."TRANSFER BUFF"."MFG TO STORAGE-3 WITH INLINE HOMO", in2 := 5)
      { S7_Templates := "SrcType := Int" } NE_Contact(in1 := "CONTINUE DB"."SYRUP MFG PROCESS ERROR", in2 := 1)
      { S7_Templates := "time_type := Time" } "IEC_Timer_0_DB_73".TON(pt := T#2S, et =>)
      Move(in := 10, out1 => "MFG TRANSFER CYCLE DB".TRANSFER."TRANSFER BUFF"."MFG TO STORAGE-3 WITH INLINE HOMO")
   END_RUNG
   // the same network as SCL:
   "IEC_Timer_0_DB_73".TON(IN := "AlwaysTRUE" AND ("MODE SELECTION DB"."MODE BUFF" = 1) AND ("MFG PROCESS_DB"."AUTO BUFF" = 0) AND ("MFG TRANSFER CYCLE DB".TRANSFER."TRANSFER BUFF"."MFG TO STORAGE-3 WITH INLINE HOMO" = 5) AND ("CONTINUE DB"."SYRUP MFG PROCESS ERROR" <> 1),
                           PT := T#2S);
   IF "IEC_Timer_0_DB_73".Q THEN
       "MFG TRANSFER CYCLE DB".TRANSFER."TRANSFER BUFF"."MFG TO STORAGE-3 WITH INLINE HOMO" := 10;
   END_IF;
END_REGION

REGION Network 33: LOAD CELL CUTOUT
   RUNG wire#powerrail
      Contact( "AlwaysTRUE" )
      { S7_Templates := "SrcType := Int" } EQ_Contact(in1 := "MODE SELECTION DB"."MODE BUFF", in2 := 1)
      { S7_Templates := "SrcType := Int" } EQ_Contact(in1 := "MFG PROCESS_DB"."AUTO BUFF", in2 := 0)
      { S7_Templates := "SrcType := Int" } EQ_Contact(in1 := "MFG TRANSFER CYCLE DB".TRANSFER."TRANSFER BUFF"."MFG TO STORAGE-3 WITH INLINE HOMO", in2 := 10)
      { S7_Templates := "SrcType := Int" } NE_Contact(in1 := "CONTINUE DB"."SYRUP MFG PROCESS ERROR", in2 := 1)
      { S7_Templates := "SrcType := Int" } EQ_Contact(in1 := "LEVEL BUFF"."SYRUP MFG_LOAD CELL", in2 := 1)
      Move(in := 15, out1 => "MFG TRANSFER CYCLE DB".TRANSFER."TRANSFER BUFF"."MFG TO STORAGE-3 WITH INLINE HOMO")
   END_RUNG
   // the same network as SCL:
   IF "AlwaysTRUE" AND ("MODE SELECTION DB"."MODE BUFF" = 1) AND ("MFG PROCESS_DB"."AUTO BUFF" = 0) AND ("MFG TRANSFER CYCLE DB".TRANSFER."TRANSFER BUFF"."MFG TO STORAGE-3 WITH INLINE HOMO" = 10) AND ("CONTINUE DB"."SYRUP MFG PROCESS ERROR" <> 1) AND ("LEVEL BUFF"."SYRUP MFG_LOAD CELL" = 1) THEN
       "MFG TRANSFER CYCLE DB".TRANSFER."TRANSFER BUFF"."MFG TO STORAGE-3 WITH INLINE HOMO" := 15;
   END_IF;
END_REGION

REGION Network 34: TIMER
   RUNG wire#powerrail
      "TIMER_SEC_DB_9"(RESET := wire#w1, INPUT := wire#w2, "SET TIME" := "MFG TRANSFER CYCLE DB"."SET PARAMETER"."SET TIME"."MFG TO STORAGE-3 WITH INLINE HOMO", "PRESENT VALUE OF TIME" => "MFG TRANSFER CYCLE DB"."PV PARAMETER"."PV TIME"."MFG TO STORAGE-3 WITH INLINE HOMO", DONE =>)
   END_RUNG
   RUNG wire#powerrail
      { S7_Templates := "SrcType := Int" } NE_Contact(in1 := "MFG TRANSFER CYCLE DB".TRANSFER."TRANSFER BUFF"."MFG TO STORAGE-3 WITH INLINE HOMO", in2 := 10)
   END_RUNG wire#w1
   RUNG wire#powerrail
      Contact( "AlwaysTRUE" )
      { S7_Templates := "SrcType := Int" } EQ_Contact(in1 := "MODE SELECTION DB"."MODE BUFF", in2 := 1)
      { S7_Templates := "SrcType := Int" } EQ_Contact(in1 := "MFG TRANSFER CYCLE DB".TRANSFER."TRANSFER BUFF"."MFG TO STORAGE-3 WITH INLINE HOMO", in2 := 10)
      { S7_Templates := "SrcType := Int" } NE_Contact(in1 := "CONTINUE DB"."SYRUP MFG PROCESS ERROR", in2 := 1)
   END_RUNG wire#w2
   // the same network as SCL:
   "TIMER_SEC_DB_9"("SET TIME" := "MFG TRANSFER CYCLE DB"."SET PARAMETER"."SET TIME"."MFG TO STORAGE-3 WITH INLINE HOMO",   // "TIMER_SEC"
                    RESET := "MFG TRANSFER CYCLE DB".TRANSFER."TRANSFER BUFF"."MFG TO STORAGE-3 WITH INLINE HOMO" <> 10,
                    INPUT := "AlwaysTRUE" AND ("MODE SELECTION DB"."MODE BUFF" = 1) AND ("MFG TRANSFER CYCLE DB".TRANSFER."TRANSFER BUFF"."MFG TO STORAGE-3 WITH INLINE HOMO" = 10) AND ("CONTINUE DB"."SYRUP MFG PROCESS ERROR" <> 1),
                    "PRESENT VALUE OF TIME" => "MFG TRANSFER CYCLE DB"."PV PARAMETER"."PV TIME"."MFG TO STORAGE-3 WITH INLINE HOMO");
END_REGION

REGION Network 35: TRANSFER OVER
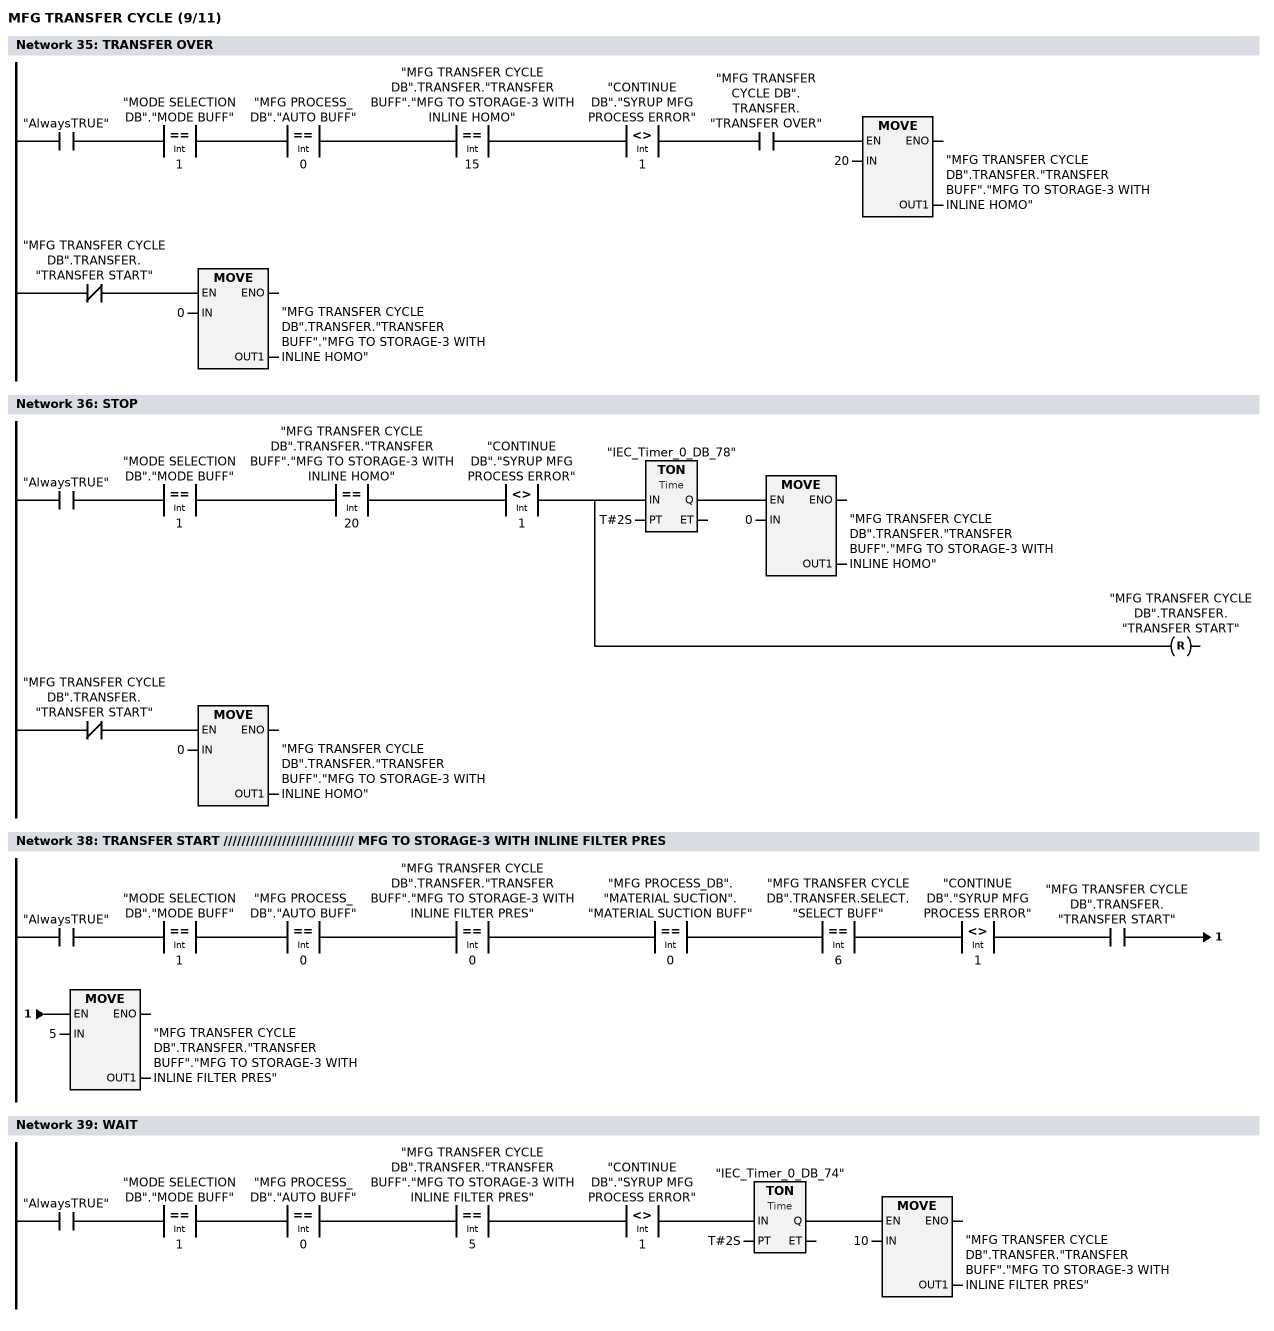
   RUNG wire#powerrail
      Contact( "AlwaysTRUE" )
      { S7_Templates := "SrcType := Int" } EQ_Contact(in1 := "MODE SELECTION DB"."MODE BUFF", in2 := 1)
      { S7_Templates := "SrcType := Int" } EQ_Contact(in1 := "MFG PROCESS_DB"."AUTO BUFF", in2 := 0)
      { S7_Templates := "SrcType := Int" } EQ_Contact(in1 := "MFG TRANSFER CYCLE DB".TRANSFER."TRANSFER BUFF"."MFG TO STORAGE-3 WITH INLINE HOMO", in2 := 15)
      { S7_Templates := "SrcType := Int" } NE_Contact(in1 := "CONTINUE DB"."SYRUP MFG PROCESS ERROR", in2 := 1)
      Contact( "MFG TRANSFER CYCLE DB".TRANSFER."TRANSFER OVER" )
      Move(in := 20, out1 => "MFG TRANSFER CYCLE DB".TRANSFER."TRANSFER BUFF"."MFG TO STORAGE-3 WITH INLINE HOMO")
   END_RUNG
   RUNG wire#powerrail
      I_Contact( "MFG TRANSFER CYCLE DB".TRANSFER."TRANSFER START" )
      Move(in := 0, out1 => "MFG TRANSFER CYCLE DB".TRANSFER."TRANSFER BUFF"."MFG TO STORAGE-3 WITH INLINE HOMO")
   END_RUNG
   // the same network as SCL:
   IF "AlwaysTRUE" AND ("MODE SELECTION DB"."MODE BUFF" = 1) AND ("MFG PROCESS_DB"."AUTO BUFF" = 0) AND ("MFG TRANSFER CYCLE DB".TRANSFER."TRANSFER BUFF"."MFG TO STORAGE-3 WITH INLINE HOMO" = 15) AND ("CONTINUE DB"."SYRUP MFG PROCESS ERROR" <> 1) AND "MFG TRANSFER CYCLE DB".TRANSFER."TRANSFER OVER" THEN
       "MFG TRANSFER CYCLE DB".TRANSFER."TRANSFER BUFF"."MFG TO STORAGE-3 WITH INLINE HOMO" := 20;
   END_IF;
   IF NOT "MFG TRANSFER CYCLE DB".TRANSFER."TRANSFER START" THEN
       "MFG TRANSFER CYCLE DB".TRANSFER."TRANSFER BUFF"."MFG TO STORAGE-3 WITH INLINE HOMO" := 0;
   END_IF;
END_REGION

REGION Network 36: STOP
   RUNG wire#powerrail
      Contact( "AlwaysTRUE" )
      { S7_Templates := "SrcType := Int" } EQ_Contact(in1 := "MODE SELECTION DB"."MODE BUFF", in2 := 1)
      { S7_Templates := "SrcType := Int" } EQ_Contact(in1 := "MFG TRANSFER CYCLE DB".TRANSFER."TRANSFER BUFF"."MFG TO STORAGE-3 WITH INLINE HOMO", in2 := 20)
      { S7_Templates := "SrcType := Int" } NE_Contact(in1 := "CONTINUE DB"."SYRUP MFG PROCESS ERROR", in2 := 1)
      wire#w1
      { S7_Templates := "time_type := Time" } "IEC_Timer_0_DB_78".TON(pt := T#2S, et =>)
      Move(in := 0, out1 => "MFG TRANSFER CYCLE DB".TRANSFER."TRANSFER BUFF"."MFG TO STORAGE-3 WITH INLINE HOMO")
   END_RUNG
   RUNG wire#w1
      R_Coil( "MFG TRANSFER CYCLE DB".TRANSFER."TRANSFER START" )
   END_RUNG
   RUNG wire#powerrail
      I_Contact( "MFG TRANSFER CYCLE DB".TRANSFER."TRANSFER START" )
      Move(in := 0, out1 => "MFG TRANSFER CYCLE DB".TRANSFER."TRANSFER BUFF"."MFG TO STORAGE-3 WITH INLINE HOMO")
   END_RUNG
   // the same network as SCL:
   #_w1 := "AlwaysTRUE" AND ("MODE SELECTION DB"."MODE BUFF" = 1) AND ("MFG TRANSFER CYCLE DB".TRANSFER."TRANSFER BUFF"."MFG TO STORAGE-3 WITH INLINE HOMO" = 20) AND ("CONTINUE DB"."SYRUP MFG PROCESS ERROR" <> 1);
   "IEC_Timer_0_DB_78".TON(IN := #_w1, PT := T#2S);
   IF "IEC_Timer_0_DB_78".Q THEN
       "MFG TRANSFER CYCLE DB".TRANSFER."TRANSFER BUFF"."MFG TO STORAGE-3 WITH INLINE HOMO" := 0;
   END_IF;
   IF #_w1 THEN "MFG TRANSFER CYCLE DB".TRANSFER."TRANSFER START" := FALSE; END_IF;
   IF NOT "MFG TRANSFER CYCLE DB".TRANSFER."TRANSFER START" THEN
       "MFG TRANSFER CYCLE DB".TRANSFER."TRANSFER BUFF"."MFG TO STORAGE-3 WITH INLINE HOMO" := 0;
   END_IF;
END_REGION

REGION Network 38: TRANSFER START ///////////////////////////// MFG TO STORAGE-3 WITH INLINE FILTER PRES
   RUNG wire#powerrail
      Contact( "AlwaysTRUE" )
      { S7_Templates := "SrcType := Int" } EQ_Contact(in1 := "MODE SELECTION DB"."MODE BUFF", in2 := 1)
      { S7_Templates := "SrcType := Int" } EQ_Contact(in1 := "MFG PROCESS_DB"."AUTO BUFF", in2 := 0)
      { S7_Templates := "SrcType := Int" } EQ_Contact(in1 := "MFG TRANSFER CYCLE DB".TRANSFER."TRANSFER BUFF"."MFG TO STORAGE-3 WITH INLINE FILTER PRES", in2 := 0)
      { S7_Templates := "SrcType := Int" } EQ_Contact(in1 := "MFG PROCESS_DB"."MATERIAL SUCTION"."MATERIAL SUCTION BUFF", in2 := 0)
      { S7_Templates := "SrcType := Int" } EQ_Contact(in1 := "MFG TRANSFER CYCLE DB".TRANSFER.SELECT."SELECT BUFF", in2 := 6)
      { S7_Templates := "SrcType := Int" } NE_Contact(in1 := "CONTINUE DB"."SYRUP MFG PROCESS ERROR", in2 := 1)
      Contact( "MFG TRANSFER CYCLE DB".TRANSFER."TRANSFER START" )
      Move(in := 5, out1 => "MFG TRANSFER CYCLE DB".TRANSFER."TRANSFER BUFF"."MFG TO STORAGE-3 WITH INLINE FILTER PRES")
   END_RUNG
   // the same network as SCL:
   IF "AlwaysTRUE" AND ("MODE SELECTION DB"."MODE BUFF" = 1) AND ("MFG PROCESS_DB"."AUTO BUFF" = 0) AND ("MFG TRANSFER CYCLE DB".TRANSFER."TRANSFER BUFF"."MFG TO STORAGE-3 WITH INLINE FILTER PRES" = 0) AND ("MFG PROCESS_DB"."MATERIAL SUCTION"."MATERIAL SUCTION BUFF" = 0) AND ("MFG TRANSFER CYCLE DB".TRANSFER.SELECT."SELECT BUFF" = 6) AND ("CONTINUE DB"."SYRUP MFG PROCESS ERROR" <> 1) AND "MFG TRANSFER CYCLE DB".TRANSFER."TRANSFER START" THEN
       "MFG TRANSFER CYCLE DB".TRANSFER."TRANSFER BUFF"."MFG TO STORAGE-3 WITH INLINE FILTER PRES" := 5;
   END_IF;
END_REGION

REGION Network 39: WAIT
   RUNG wire#powerrail
      Contact( "AlwaysTRUE" )
      { S7_Templates := "SrcType := Int" } EQ_Contact(in1 := "MODE SELECTION DB"."MODE BUFF", in2 := 1)
      { S7_Templates := "SrcType := Int" } EQ_Contact(in1 := "MFG PROCESS_DB"."AUTO BUFF", in2 := 0)
      { S7_Templates := "SrcType := Int" } EQ_Contact(in1 := "MFG TRANSFER CYCLE DB".TRANSFER."TRANSFER BUFF"."MFG TO STORAGE-3 WITH INLINE FILTER PRES", in2 := 5)
      { S7_Templates := "SrcType := Int" } NE_Contact(in1 := "CONTINUE DB"."SYRUP MFG PROCESS ERROR", in2 := 1)
      { S7_Templates := "time_type := Time" } "IEC_Timer_0_DB_74".TON(pt := T#2S, et =>)
      Move(in := 10, out1 => "MFG TRANSFER CYCLE DB".TRANSFER."TRANSFER BUFF"."MFG TO STORAGE-3 WITH INLINE FILTER PRES")
   END_RUNG
   // the same network as SCL:
   "IEC_Timer_0_DB_74".TON(IN := "AlwaysTRUE" AND ("MODE SELECTION DB"."MODE BUFF" = 1) AND ("MFG PROCESS_DB"."AUTO BUFF" = 0) AND ("MFG TRANSFER CYCLE DB".TRANSFER."TRANSFER BUFF"."MFG TO STORAGE-3 WITH INLINE FILTER PRES" = 5) AND ("CONTINUE DB"."SYRUP MFG PROCESS ERROR" <> 1),
                           PT := T#2S);
   IF "IEC_Timer_0_DB_74".Q THEN
       "MFG TRANSFER CYCLE DB".TRANSFER."TRANSFER BUFF"."MFG TO STORAGE-3 WITH INLINE FILTER PRES" := 10;
   END_IF;
END_REGION

REGION Network 40: LOAD CELL CUTOUT
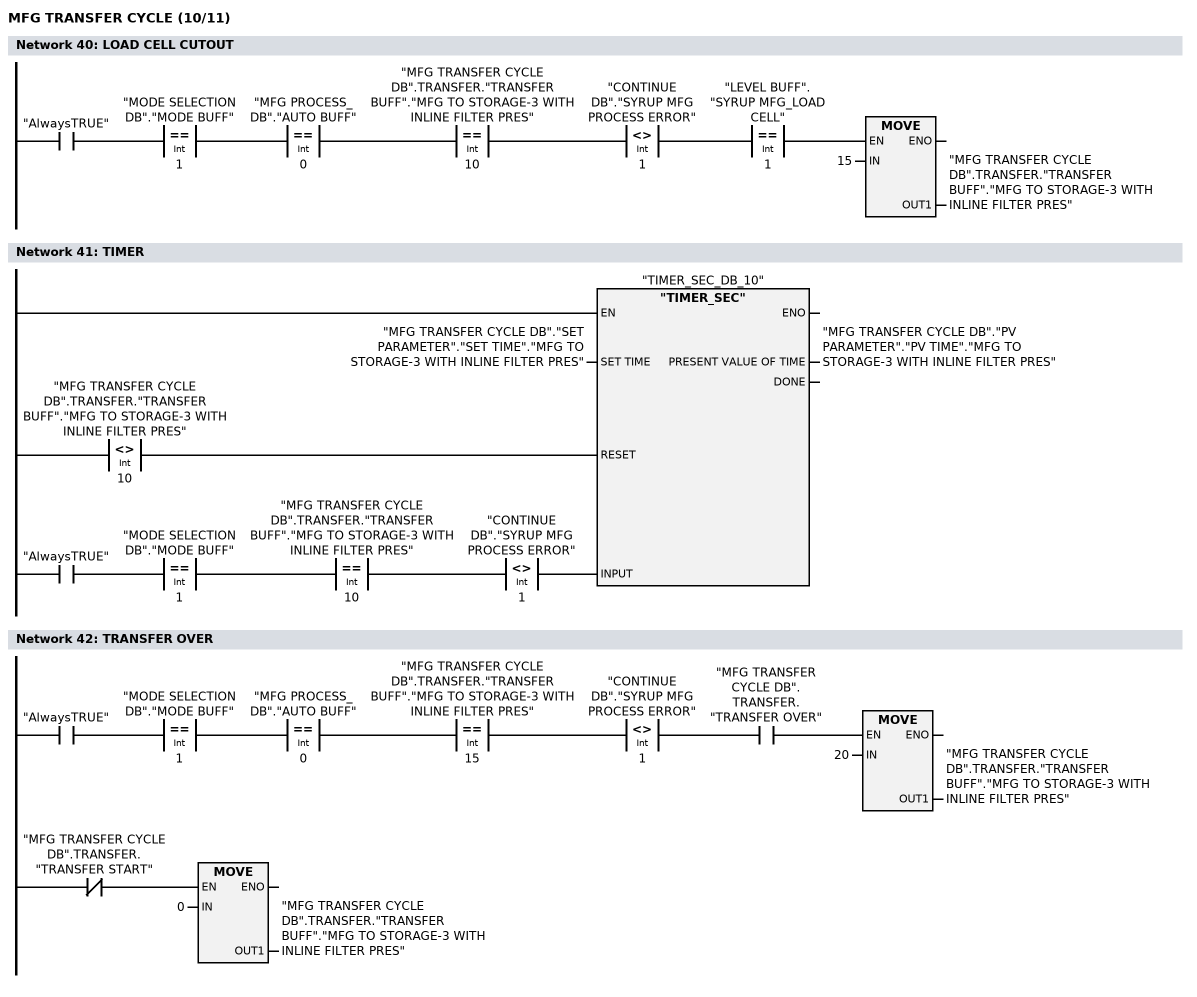
   RUNG wire#powerrail
      Contact( "AlwaysTRUE" )
      { S7_Templates := "SrcType := Int" } EQ_Contact(in1 := "MODE SELECTION DB"."MODE BUFF", in2 := 1)
      { S7_Templates := "SrcType := Int" } EQ_Contact(in1 := "MFG PROCESS_DB"."AUTO BUFF", in2 := 0)
      { S7_Templates := "SrcType := Int" } EQ_Contact(in1 := "MFG TRANSFER CYCLE DB".TRANSFER."TRANSFER BUFF"."MFG TO STORAGE-3 WITH INLINE FILTER PRES", in2 := 10)
      { S7_Templates := "SrcType := Int" } NE_Contact(in1 := "CONTINUE DB"."SYRUP MFG PROCESS ERROR", in2 := 1)
      { S7_Templates := "SrcType := Int" } EQ_Contact(in1 := "LEVEL BUFF"."SYRUP MFG_LOAD CELL", in2 := 1)
      Move(in := 15, out1 => "MFG TRANSFER CYCLE DB".TRANSFER."TRANSFER BUFF"."MFG TO STORAGE-3 WITH INLINE FILTER PRES")
   END_RUNG
   // the same network as SCL:
   IF "AlwaysTRUE" AND ("MODE SELECTION DB"."MODE BUFF" = 1) AND ("MFG PROCESS_DB"."AUTO BUFF" = 0) AND ("MFG TRANSFER CYCLE DB".TRANSFER."TRANSFER BUFF"."MFG TO STORAGE-3 WITH INLINE FILTER PRES" = 10) AND ("CONTINUE DB"."SYRUP MFG PROCESS ERROR" <> 1) AND ("LEVEL BUFF"."SYRUP MFG_LOAD CELL" = 1) THEN
       "MFG TRANSFER CYCLE DB".TRANSFER."TRANSFER BUFF"."MFG TO STORAGE-3 WITH INLINE FILTER PRES" := 15;
   END_IF;
END_REGION

REGION Network 41: TIMER
   RUNG wire#powerrail
      "TIMER_SEC_DB_10"(RESET := wire#w1, INPUT := wire#w2, "SET TIME" := "MFG TRANSFER CYCLE DB"."SET PARAMETER"."SET TIME"."MFG TO STORAGE-3 WITH INLINE FILTER PRES", "PRESENT VALUE OF TIME" => "MFG TRANSFER CYCLE DB"."PV PARAMETER"."PV TIME"."MFG TO STORAGE-3 WITH INLINE FILTER PRES", DONE =>)
   END_RUNG
   RUNG wire#powerrail
      { S7_Templates := "SrcType := Int" } NE_Contact(in1 := "MFG TRANSFER CYCLE DB".TRANSFER."TRANSFER BUFF"."MFG TO STORAGE-3 WITH INLINE FILTER PRES", in2 := 10)
   END_RUNG wire#w1
   RUNG wire#powerrail
      Contact( "AlwaysTRUE" )
      { S7_Templates := "SrcType := Int" } EQ_Contact(in1 := "MODE SELECTION DB"."MODE BUFF", in2 := 1)
      { S7_Templates := "SrcType := Int" } EQ_Contact(in1 := "MFG TRANSFER CYCLE DB".TRANSFER."TRANSFER BUFF"."MFG TO STORAGE-3 WITH INLINE FILTER PRES", in2 := 10)
      { S7_Templates := "SrcType := Int" } NE_Contact(in1 := "CONTINUE DB"."SYRUP MFG PROCESS ERROR", in2 := 1)
   END_RUNG wire#w2
   // the same network as SCL:
   "TIMER_SEC_DB_10"("SET TIME" := "MFG TRANSFER CYCLE DB"."SET PARAMETER"."SET TIME"."MFG TO STORAGE-3 WITH INLINE FILTER PRES",   // "TIMER_SEC"
                     RESET := "MFG TRANSFER CYCLE DB".TRANSFER."TRANSFER BUFF"."MFG TO STORAGE-3 WITH INLINE FILTER PRES" <> 10,
                     INPUT := "AlwaysTRUE" AND ("MODE SELECTION DB"."MODE BUFF" = 1) AND ("MFG TRANSFER CYCLE DB".TRANSFER."TRANSFER BUFF"."MFG TO STORAGE-3 WITH INLINE FILTER PRES" = 10) AND ("CONTINUE DB"."SYRUP MFG PROCESS ERROR" <> 1),
                     "PRESENT VALUE OF TIME" => "MFG TRANSFER CYCLE DB"."PV PARAMETER"."PV TIME"."MFG TO STORAGE-3 WITH INLINE FILTER PRES");
END_REGION

REGION Network 42: TRANSFER OVER
   RUNG wire#powerrail
      Contact( "AlwaysTRUE" )
      { S7_Templates := "SrcType := Int" } EQ_Contact(in1 := "MODE SELECTION DB"."MODE BUFF", in2 := 1)
      { S7_Templates := "SrcType := Int" } EQ_Contact(in1 := "MFG PROCESS_DB"."AUTO BUFF", in2 := 0)
      { S7_Templates := "SrcType := Int" } EQ_Contact(in1 := "MFG TRANSFER CYCLE DB".TRANSFER."TRANSFER BUFF"."MFG TO STORAGE-3 WITH INLINE FILTER PRES", in2 := 15)
      { S7_Templates := "SrcType := Int" } NE_Contact(in1 := "CONTINUE DB"."SYRUP MFG PROCESS ERROR", in2 := 1)
      Contact( "MFG TRANSFER CYCLE DB".TRANSFER."TRANSFER OVER" )
      Move(in := 20, out1 => "MFG TRANSFER CYCLE DB".TRANSFER."TRANSFER BUFF"."MFG TO STORAGE-3 WITH INLINE FILTER PRES")
   END_RUNG
   RUNG wire#powerrail
      I_Contact( "MFG TRANSFER CYCLE DB".TRANSFER."TRANSFER START" )
      Move(in := 0, out1 => "MFG TRANSFER CYCLE DB".TRANSFER."TRANSFER BUFF"."MFG TO STORAGE-3 WITH INLINE FILTER PRES")
   END_RUNG
   // the same network as SCL:
   IF "AlwaysTRUE" AND ("MODE SELECTION DB"."MODE BUFF" = 1) AND ("MFG PROCESS_DB"."AUTO BUFF" = 0) AND ("MFG TRANSFER CYCLE DB".TRANSFER."TRANSFER BUFF"."MFG TO STORAGE-3 WITH INLINE FILTER PRES" = 15) AND ("CONTINUE DB"."SYRUP MFG PROCESS ERROR" <> 1) AND "MFG TRANSFER CYCLE DB".TRANSFER."TRANSFER OVER" THEN
       "MFG TRANSFER CYCLE DB".TRANSFER."TRANSFER BUFF"."MFG TO STORAGE-3 WITH INLINE FILTER PRES" := 20;
   END_IF;
   IF NOT "MFG TRANSFER CYCLE DB".TRANSFER."TRANSFER START" THEN
       "MFG TRANSFER CYCLE DB".TRANSFER."TRANSFER BUFF"."MFG TO STORAGE-3 WITH INLINE FILTER PRES" := 0;
   END_IF;
END_REGION

REGION Network 43: STOP
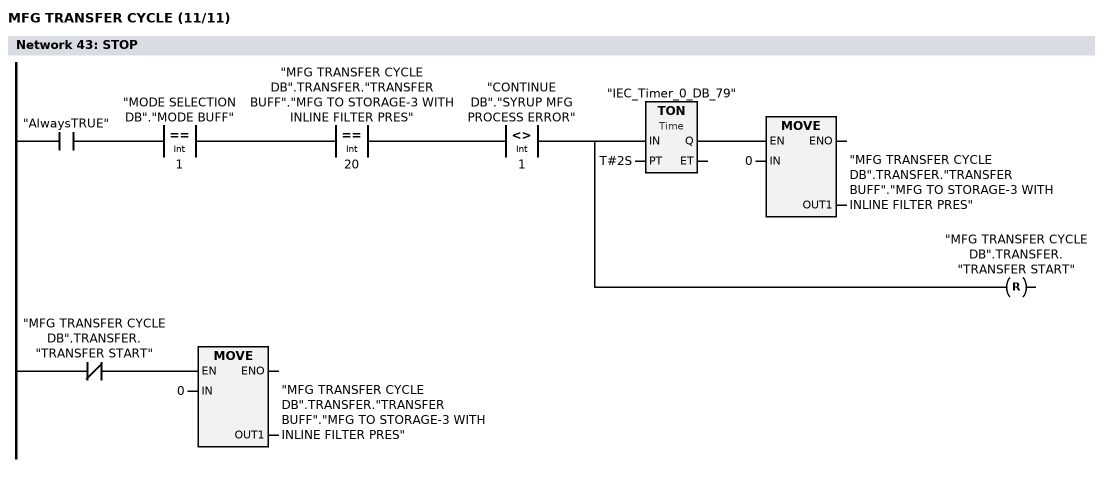
   RUNG wire#powerrail
      Contact( "AlwaysTRUE" )
      { S7_Templates := "SrcType := Int" } EQ_Contact(in1 := "MODE SELECTION DB"."MODE BUFF", in2 := 1)
      { S7_Templates := "SrcType := Int" } EQ_Contact(in1 := "MFG TRANSFER CYCLE DB".TRANSFER."TRANSFER BUFF"."MFG TO STORAGE-3 WITH INLINE FILTER PRES", in2 := 20)
      { S7_Templates := "SrcType := Int" } NE_Contact(in1 := "CONTINUE DB"."SYRUP MFG PROCESS ERROR", in2 := 1)
      wire#w1
      { S7_Templates := "time_type := Time" } "IEC_Timer_0_DB_79".TON(pt := T#2S, et =>)
      Move(in := 0, out1 => "MFG TRANSFER CYCLE DB".TRANSFER."TRANSFER BUFF"."MFG TO STORAGE-3 WITH INLINE FILTER PRES")
   END_RUNG
   RUNG wire#w1
      R_Coil( "MFG TRANSFER CYCLE DB".TRANSFER."TRANSFER START" )
   END_RUNG
   RUNG wire#powerrail
      I_Contact( "MFG TRANSFER CYCLE DB".TRANSFER."TRANSFER START" )
      Move(in := 0, out1 => "MFG TRANSFER CYCLE DB".TRANSFER."TRANSFER BUFF"."MFG TO STORAGE-3 WITH INLINE FILTER PRES")
   END_RUNG
   // the same network as SCL:
   #_w1 := "AlwaysTRUE" AND ("MODE SELECTION DB"."MODE BUFF" = 1) AND ("MFG TRANSFER CYCLE DB".TRANSFER."TRANSFER BUFF"."MFG TO STORAGE-3 WITH INLINE FILTER PRES" = 20) AND ("CONTINUE DB"."SYRUP MFG PROCESS ERROR" <> 1);
   "IEC_Timer_0_DB_79".TON(IN := #_w1, PT := T#2S);
   IF "IEC_Timer_0_DB_79".Q THEN
       "MFG TRANSFER CYCLE DB".TRANSFER."TRANSFER BUFF"."MFG TO STORAGE-3 WITH INLINE FILTER PRES" := 0;
   END_IF;
   IF #_w1 THEN "MFG TRANSFER CYCLE DB".TRANSFER."TRANSFER START" := FALSE; END_IF;
   IF NOT "MFG TRANSFER CYCLE DB".TRANSFER."TRANSFER START" THEN
       "MFG TRANSFER CYCLE DB".TRANSFER."TRANSFER BUFF"."MFG TO STORAGE-3 WITH INLINE FILTER PRES" := 0;
   END_IF;
END_REGION
END_FUNCTION
